KUKA KRL program: EPS_2_251825_SA26_A_20260116064103.src

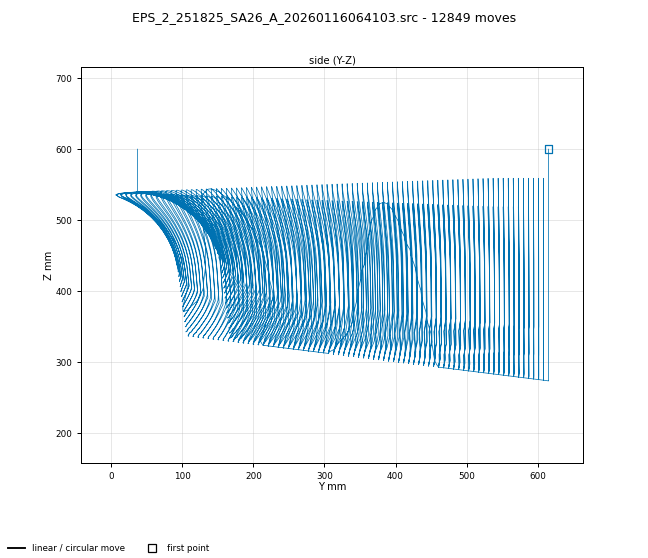
[picture p0: tool path of EPS_2_251825_SA26_A_20260116064103.src, 12849 of 12851 moves have a stored position in this frame; points joined in program order, loops and branches not executed]
&ACCESS RVP
&REL 4
&COMMENT QRS 19112012
&PARAM EDITMASK = *
DEF PART()
EXT BAS (BAS_COMMAND :IN,REAL :IN )
INT I
BAS (#INITMOV,0 )

;KUKA QRS Post kuka4.cps  Date:22-06-2017 !

File_ID=2985

QRS_PRE_INIT()

;Init var - Until changes are made in qrs_pre_init
Outlet_Square_prg=0
Inlet_1_Square_prg=0
Inlet_2_Square_prg=0
Inlet_3_Square_prg=0
Inlet_4_Square_prg=0
Inlet_5_Square_prg=0

Outlet_1={X 0.000, Y 535.490, Z 458.500, B 0.000, E1 0.000 }
Inlet_1={X 0.000, Y 538.340, Z 418.500, B 0.000, E1 190.000 }
Outlet_1_type=201
Inlet_1_type=201
;QRS#1=Sidecore dimensions
;QRS#2=200-8" PVC SDR 35
;QRS#3=200-8" PVC SDR 35
;QRS#4=
;QRS#5=
;QRS#6=
;QRS#7=
;QRS#8=
;QRS#9=12-08 PSX
;QRS#10=12-08 PSX
;QRS#11=
;QRS#12=
;QRS#13=
;QRS#14=
;QRS#15=
;QRS#16=1220x127x838 2,75'
;QRS#17=EPS Height
;QRS#18=559
;QRS#19=*
;QRS#20= UPDATED VERSION 22-06-2017
;QRS#21=*
Outlet_Square=0100
Inlet_1_Square=0100
Inlet_2_Square=0
Inlet_3_Square=0
Inlet_4_Square=0
Inlet_5_Square=0
Mill_Square=1
Outlet_Square_Prg=204
Inlet_1_Square_prg=204

QRS_INIT()

$ADVANCE=5

; T1
PTP {E1 173.626,E2 173.626}
PTP {X 0,Y 615.464,A -85,B 0,C 180,E1 173.626,E2 173.626,E3 0,E4 0,E5 0,E6 0}
QRS_SPEED_INIT()
LIN {X 0,Y 615.464,Z 600,A -85,B 0,C 180,E1 173.626,E2 173.626,E3 0,E4 0,E5 0,E6 0} C_VEL
LIN {X 0,Y 615.464,Z 283.872,A -85,B 0,C 180,E1 173.626,E2 173.626} C_VEL
LIN {X 0,Y 615.464,Z 275.69,A -85,B 0,C 180,E1 173.626,E2 173.626} C_VEL
LIN {X 0,Y 615.457,Z 273.69,A -85,B 0,C 180,E1 173.44,E2 173.44} C_VEL
LIN {X 0,Y 615.487,Z 273.682,A -85,B 0,C 180,E1 170.801,E2 170.801} C_VEL
LIN {X 0,Y 615.491,Z 273.695,A -85,B 0,C 180,E1 168.139,E2 168.139} C_VEL
LIN {X 0,Y 615.461,Z 273.694,A -85,B 0,C 180,E1 165.45,E2 165.45} C_VEL
LIN {X 0,Y 615.46,Z 273.695,A -85,B 0,C 180,E1 163.413,E2 163.413} C_VEL
LIN {X 0,Y 615.46,Z 273.694,A -85,B 0,C 180,E1 161.353,E2 161.353} C_VEL
LIN {X 0,Y 615.458,Z 273.694,A -85,B 0,C 180,E1 159.268,E2 159.268} C_VEL
LIN {X 0,Y 615.455,Z 273.694,A -85,B 0,C 180,E1 157.154,E2 157.154} C_VEL
LIN {X 0,Y 615.451,Z 273.693,A -85,B 0,C 180,E1 155.007,E2 155.007} C_VEL
LIN {X 0,Y 615.449,Z 273.691,A -85,B 0,C 180,E1 152.821,E2 152.821} C_VEL
LIN {X 0,Y 615.476,Z 273.685,A -85,B 0,C 180,E1 150.206,E2 150.206} C_VEL
LIN {X 0,Y 615.493,Z 273.695,A -85,B 0,C 180,E1 147.543,E2 147.543} C_VEL
LIN {X 0,Y 615.482,Z 273.698,A -85,B 0,C 180,E1 145.185,E2 145.185} C_VEL
LIN {X 0,Y 615.45,Z 273.695,A -85,B 0,C 180,E1 142.755,E2 142.755} C_VEL
LIN {X 0,Y 615.447,Z 273.69,A -85,B 0,C 180,E1 140.247,E2 140.247} C_VEL
LIN {X 0,Y 615.491,Z 273.685,A -85,B 0,C 180,E1 137.647,E2 137.647} C_VEL
LIN {X 0,Y 615.484,Z 273.699,A -85,B 0,C 180,E1 134.931,E2 134.931} C_VEL
LIN {X 0,Y 615.442,Z 273.694,A -85,B 0,C 180,E1 132.356,E2 132.356} C_VEL
LIN {X 0,Y 615.439,Z 273.692,A -85,B 0,C 180,E1 130.084,E2 130.084} C_VEL
LIN {X 0,Y 615.438,Z 273.692,A -85,B 0,C 180,E1 128.006,E2 128.006} C_VEL
LIN {X 0,Y 615.449,Z 273.69,A -85,B 0,C 180,E1 125.618,E2 125.618} C_VEL
LIN {X 0,Y 615.474,Z 273.689,A -85,B 0,C 180,E1 123.236,E2 123.236} C_VEL
LIN {X 0,Y 615.49,Z 273.692,A -85,B 0,C 180,E1 120.919,E2 120.919} C_VEL
LIN {X 0,Y 615.435,Z 273.695,A -85,B 0,C 180,E1 117.917,E2 117.917} C_VEL
LIN {X 0,Y 615.433,Z 273.693,A -85,B 0,C 180,E1 115.558,E2 115.558} C_VEL
LIN {X 0,Y 615.484,Z 273.689,A -85,B 0,C 180,E1 112.844,E2 112.844} C_VEL
LIN {X 0,Y 615.455,Z 273.698,A -85,B 0,C 180,E1 110.033,E2 110.033} C_VEL
LIN {X 0,Y 615.453,Z 273.698,A -85,B 0,C 180,E1 107.958,E2 107.958} C_VEL
LIN {X 0,Y 615.452,Z 273.698,A -85,B 0,C 180,E1 105.906,E2 105.906} C_VEL
LIN {X 0,Y 615.455,Z 273.698,A -85,B 0,C 180,E1 103.875,E2 103.875} C_VEL
LIN {X 0,Y 615.46,Z 273.699,A -85,B 0,C 180,E1 101.861,E2 101.861} C_VEL
LIN {X 0,Y 615.423,Z 273.696,A -85,B 0,C 180,E1 99.199,E2 99.199} C_VEL
LIN {X 0,Y 615.453,Z 273.715,A -85,B 0,C 180,E1 98.62,E2 98.62} C_VEL
LIN {X 0,Y 615.457,Z 289.755,A -85,B 0,C 180,E1 95.899,E2 95.899} C_VEL
LIN {X 0,Y 615.446,Z 303.472,A -85,B 0,C 180,E1 93.601,E2 93.601} C_VEL
LIN {X 0,Y 615.464,Z 308.129,A -85,B 0,C 180,E1 92.822,E2 92.822} C_VEL
LIN {X 0,Y 615.458,Z 415.467,A -85,B 0,C 180,E1 91.533,E2 91.533} C_VEL
LIN {X 0,Y 615.458,Z 429.062,A -85,B 0,C 180,E1 91.227,E2 91.227} C_VEL
LIN {X 0,Y 615.485,Z 441.275,A -85,B 0,C 180,E1 90.818,E2 90.818} C_VEL
LIN {X 0,Y 615.489,Z 452.256,A -85,B 0,C 180,E1 90.327,E2 90.327} C_VEL
LIN {X 0,Y 615.488,Z 463.666,A -85,B 0,C 180,E1 89.673,E2 89.673} C_VEL
LIN {X 0,Y 615.499,Z 473.94,A -85,B 0,C 180,E1 88.937,E2 88.937} C_VEL
LIN {X 0,Y 615.497,Z 482.288,A -85,B 0,C 180,E1 88.2,E2 88.2} C_VEL
LIN {X 0,Y 615.497,Z 490.195,A -85,B 0,C 180,E1 87.382,E2 87.382} C_VEL
LIN {X 0,Y 615.493,Z 497.851,A -85,B 0,C 180,E1 86.399,E2 86.399} C_VEL
LIN {X 0,Y 615.496,Z 504.004,A -85,B 0,C 180,E1 85.415,E2 85.415} C_VEL
LIN {X 0,Y 615.497,Z 508.911,A -85,B 0,C 180,E1 84.43,E2 84.43} C_VEL
LIN {X 0,Y 615.495,Z 512.797,A -85,B 0,C 180,E1 83.416,E2 83.416} C_VEL
LIN {X 0,Y 615.495,Z 516.218,A -85,B 0,C 180,E1 82.124,E2 82.124} C_VEL
LIN {X 0,Y 615.495,Z 517.345,A -85,B 0,C 180,E1 81.463,E2 81.463} C_VEL
LIN {X 0,Y 615.496,Z 518.351,A -85,B 0,C 180,E1 80.138,E2 80.138} C_VEL
LIN {X 0,Y 615.494,Z 518.038,A -85,B 0,C 180,E1 79.109,E2 79.109} C_VEL
LIN {X 0,Y 615.495,Z 516.853,A -85,B 0,C 180,E1 78.139,E2 78.139} C_VEL
LIN {X 0,Y 615.496,Z 515.533,A -85,B 0,C 180,E1 77.47,E2 77.47} C_VEL
LIN {X 0,Y 615.496,Z 512.696,A -85,B 0,C 180,E1 76.463,E2 76.463} C_VEL
LIN {X 0,Y 615.497,Z 508.787,A -85,B 0,C 180,E1 75.451,E2 75.451} C_VEL
LIN {X 0,Y 615.496,Z 503.676,A -85,B 0,C 180,E1 74.435,E2 74.435} C_VEL
LIN {X 0,Y 615.495,Z 497.179,A -85,B 0,C 180,E1 73.414,E2 73.414} C_VEL
LIN {X 0,Y 615.498,Z 488.929,A -85,B 0,C 180,E1 72.387,E2 72.387} C_VEL
LIN {X 0,Y 615.497,Z 478.509,A -85,B 0,C 180,E1 71.354,E2 71.354} C_VEL
LIN {X 0,Y 615.494,Z 467.446,A -85,B 0,C 180,E1 70.489,E2 70.489} C_VEL
LIN {X 0,Y 615.465,Z 457.023,A -85,B 0,C 180,E1 69.836,E2 69.836} C_VEL
LIN {X 0,Y 615.492,Z 445.516,A -85,B 0,C 180,E1 69.269,E2 69.269} C_VEL
LIN {X 0,Y 615.443,Z 432.543,A -85,B 0,C 180,E1 68.786,E2 68.786} C_VEL
LIN {X 0,Y 615.424,Z 419.82,A -85,B 0,C 180,E1 68.456,E2 68.456} C_VEL
LIN {X 0,Y 615.422,Z 405.107,A -85,B 0,C 180,E1 68.236,E2 68.236} C_VEL
LIN {X 0,Y 615.476,Z 308.131,A -85,B 0,C 180,E1 67.088,E2 67.088} C_VEL
LIN {X 0,Y 615.45,Z 292.299,A -85,B 0,C 180,E1 64.438,E2 64.438} C_VEL
LIN {X 0,Y 615.494,Z 276.796,A -85,B 0,C 180,E1 61.818,E2 61.818} C_VEL
LIN {X 0,Y 615.488,Z 273.684,A -85,B 0,C 180,E1 61.249,E2 61.249} C_VEL
LIN {X 0,Y 615.483,Z 273.682,A -85,B 0,C 180,E1 58.915,E2 58.915} C_VEL
LIN {X 0,Y 615.469,Z 273.686,A -85,B 0,C 180,E1 56.468,E2 56.468} C_VEL
LIN {X 0,Y 615.466,Z 273.69,A -85,B 0,C 180,E1 54.169,E2 54.169} C_VEL
LIN {X 0,Y 615.471,Z 273.693,A -85,B 0,C 180,E1 51.93,E2 51.93} C_VEL
LIN {X 0,Y 615.493,Z 273.698,A -85,B 0,C 180,E1 49.394,E2 49.394} C_VEL
LIN {X 0,Y 615.487,Z 273.683,A -85,B 0,C 180,E1 46.755,E2 46.755} C_VEL
LIN {X 0,Y 615.469,Z 273.687,A -85,B 0,C 180,E1 43.996,E2 43.996} C_VEL
LIN {X 0,Y 615.479,Z 273.696,A -85,B 0,C 180,E1 41.474,E2 41.474} C_VEL
LIN {X 0,Y 615.484,Z 273.694,A -85,B 0,C 180,E1 38.904,E2 38.904} C_VEL
LIN {X 0,Y 615.486,Z 273.683,A -85,B 0,C 180,E1 36.425,E2 36.425} C_VEL
LIN {X 0,Y 615.489,Z 273.68,A -85,B 0,C 180,E1 34.022,E2 34.022} C_VEL
LIN {X 0,Y 615.48,Z 273.698,A -85,B 0,C 180,E1 31.085,E2 31.085} C_VEL
LIN {X 0,Y 615.48,Z 273.69,A -85,B 0,C 180,E1 28.449,E2 28.449} C_VEL
LIN {X 0,Y 615.477,Z 273.684,A -85,B 0,C 180,E1 25.567,E2 25.567} C_VEL
LIN {X 0,Y 615.484,Z 273.697,A -85,B 0,C 180,E1 22.845,E2 22.845} C_VEL
LIN {X 0,Y 615.48,Z 273.687,A -85,B 0,C 180,E1 20.033,E2 20.033} C_VEL
LIN {X 0,Y 615.474,Z 273.685,A -85,B 0,C 180,E1 17.271,E2 17.271} C_VEL
LIN {X 0,Y 615.488,Z 273.697,A -85,B 0,C 180,E1 14.549,E2 14.549} C_VEL
LIN {X 0,Y 615.478,Z 273.689,A -85,B 0,C 180,E1 11.861,E2 11.861} C_VEL
LIN {X 0,Y 615.49,Z 273.68,A -85,B 0,C 180,E1 9.199,E2 9.199} C_VEL
LIN {X 0,Y 615.474,Z 273.692,A -85,B 0,C 180,E1 6.557,E2 6.557} C_VEL
LIN {X 0,Y 615.488,Z 273.696,A -85,B 0,C 180,E1 3.928,E2 3.928} C_VEL
LIN {X 0,Y 615.482,Z 273.684,A -85,B 0,C 180,E1 1.308,E2 1.308} C_VEL
LIN {X 0,Y 615.48,Z 273.683,A -85,B 0,C 180,E1 -1.309,E2 -1.309} C_VEL
LIN {X 0,Y 615.482,Z 273.695,A -85,B 0,C 180,E1 -3.929,E2 -3.929} C_VEL
LIN {X 0,Y 615.475,Z 273.693,A -85,B 0,C 180,E1 -6.57,E2 -6.57} C_VEL
LIN {X 0,Y 615.491,Z 273.68,A -85,B 0,C 180,E1 -9.199,E2 -9.199} C_VEL
LIN {X 0,Y 615.475,Z 273.688,A -85,B 0,C 180,E1 -11.861,E2 -11.861} C_VEL
LIN {X 0,Y 615.492,Z 273.699,A -85,B 0,C 180,E1 -14.549,E2 -14.549} C_VEL
LIN {X 0,Y 615.476,Z 273.685,A -85,B 0,C 180,E1 -17.271,E2 -17.271} C_VEL
LIN {X 0,Y 615.478,Z 273.686,A -85,B 0,C 180,E1 -20.033,E2 -20.033} C_VEL
LIN {X 0,Y 615.49,Z 273.698,A -85,B 0,C 180,E1 -22.845,E2 -22.845} C_VEL
LIN {X 0,Y 615.488,Z 273.681,A -85,B 0,C 180,E1 -25.716,E2 -25.716} C_VEL
LIN {X 0,Y 615.477,Z 273.689,A -85,B 0,C 180,E1 -28.449,E2 -28.449} C_VEL
LIN {X 0,Y 615.482,Z 273.7,A -85,B 0,C 180,E1 -31.086,E2 -31.086} C_VEL
LIN {X 0,Y 615.49,Z 273.68,A -85,B 0,C 180,E1 -34.022,E2 -34.022} C_VEL
LIN {X 0,Y 615.484,Z 273.695,A -85,B 0,C 180,E1 -36.936,E2 -36.936} C_VEL
LIN {X 0,Y 615.472,Z 273.69,A -85,B 0,C 180,E1 -39.752,E2 -39.752} C_VEL
LIN {X 0,Y 615.493,Z 273.679,A -85,B 0,C 180,E1 -42.353,E2 -42.353} C_VEL
LIN {X 0,Y 615.477,Z 273.692,A -85,B 0,C 180,E1 -45.07,E2 -45.07} C_VEL
LIN {X 0,Y 615.469,Z 273.692,A -85,B 0,C 180,E1 -47.922,E2 -47.922} C_VEL
LIN {X 0,Y 615.472,Z 273.686,A -85,B 0,C 180,E1 -50.249,E2 -50.249} C_VEL
LIN {X 0,Y 615.481,Z 273.685,A -85,B 0,C 180,E1 -53.065,E2 -53.065} C_VEL
LIN {X 0,Y 615.481,Z 273.696,A -85,B 0,C 180,E1 -55.978,E2 -55.978} C_VEL
LIN {X 0,Y 615.47,Z 273.69,A -85,B 0,C 180,E1 -58.314,E2 -58.314} C_VEL
LIN {X 0,Y 615.471,Z 273.686,A -85,B 0,C 180,E1 -60.593,E2 -60.593} C_VEL
LIN {X 0,Y 615.486,Z 273.681,A -85,B 0,C 180,E1 -62.956,E2 -62.956} C_VEL
LIN {X 0,Y 615.481,Z 273.692,A -85,B 0,C 180,E1 -65.728,E2 -65.728} C_VEL
LIN {X 0,Y 615.487,Z 273.754,A -85,B 0,C 180,E1 -67.437,E2 -67.437} C_VEL
LIN {X 0,Y 615.455,Z 293.691,A -85,B 0,C 180,E1 -70.14,E2 -70.14} C_VEL
LIN {X 0,Y 615.472,Z 313.076,A -85,B 0,C 180,E1 -72.729,E2 -72.729} C_VEL
LIN {X 0,Y 615.493,Z 334.916,A -85,B 0,C 180,E1 -75.606,E2 -75.606} C_VEL
LIN {X 0,Y 615.471,Z 346.467,A -85,B 0,C 180,E1 -77.113,E2 -77.113} C_VEL
LIN {X 0,Y 615.457,Z 454.829,A -85,B 0,C 180,E1 -78.41,E2 -78.41} C_VEL
LIN {X 0,Y 615.456,Z 467.345,A -85,B 0,C 180,E1 -78.681,E2 -78.681} C_VEL
LIN {X 0,Y 615.483,Z 480.688,A -85,B 0,C 180,E1 -79.116,E2 -79.116} C_VEL
LIN {X 0,Y 615.492,Z 492.473,A -85,B 0,C 180,E1 -79.639,E2 -79.639} C_VEL
LIN {X 0,Y 615.483,Z 503.994,A -85,B 0,C 180,E1 -80.304,E2 -80.304} C_VEL
LIN {X 0,Y 615.499,Z 514.339,A -85,B 0,C 180,E1 -81.05,E2 -81.05} C_VEL
LIN {X 0,Y 615.497,Z 522.69,A -85,B 0,C 180,E1 -81.794,E2 -81.794} C_VEL
LIN {X 0,Y 615.498,Z 530.605,A -85,B 0,C 180,E1 -82.619,E2 -82.619} C_VEL
LIN {X 0,Y 615.491,Z 538.203,A -85,B 0,C 180,E1 -83.608,E2 -83.608} C_VEL
LIN {X 0,Y 615.498,Z 545.203,A -85,B 0,C 180,E1 -84.759,E2 -84.759} C_VEL
LIN {X 0,Y 615.493,Z 549.851,A -85,B 0,C 180,E1 -85.743,E2 -85.743} C_VEL
LIN {X 0,Y 615.494,Z 553.398,A -85,B 0,C 180,E1 -86.727,E2 -86.727} C_VEL
LIN {X 0,Y 615.497,Z 555.232,A -85,B 0,C 180,E1 -87.382,E2 -87.382} C_VEL
LIN {X 0,Y 615.497,Z 556.608,A -85,B 0,C 180,E1 -88.037,E2 -88.037} C_VEL
LIN {X 0,Y 615.496,Z 558.173,A -85,B 0,C 180,E1 -89.346,E2 -89.346} C_VEL
LIN {X 0,Y 615.494,Z 558.389,A -85,B 0,C 180,E1 -90,E2 -90} C_VEL
LIN {X 0,Y 615.495,Z 557.58,A -85,B 0,C 180,E1 -91.308,E2 -91.308} C_VEL
LIN {X 0,Y 615.497,Z 556.609,A -85,B 0,C 180,E1 -91.963,E2 -91.963} C_VEL
LIN {X 0,Y 615.497,Z 555.234,A -85,B 0,C 180,E1 -92.618,E2 -92.618} C_VEL
LIN {X 0,Y 615.496,Z 552.35,A -85,B 0,C 180,E1 -93.6,E2 -93.6} C_VEL
LIN {X 0,Y 615.498,Z 548.443,A -85,B 0,C 180,E1 -94.584,E2 -94.584} C_VEL
LIN {X 0,Y 615.499,Z 543.406,A -85,B 0,C 180,E1 -95.569,E2 -95.569} C_VEL
LIN {X 0,Y 615.49,Z 536.913,A -85,B 0,C 180,E1 -96.578,E2 -96.578} C_VEL
LIN {X 0,Y 615.497,Z 529.136,A -85,B 0,C 180,E1 -97.545,E2 -97.545} C_VEL
LIN {X 0,Y 615.498,Z 519.261,A -85,B 0,C 180,E1 -98.536,E2 -98.536} C_VEL
LIN {X 0,Y 615.495,Z 508.87,A -85,B 0,C 180,E1 -99.364,E2 -99.364} C_VEL
LIN {X 0,Y 615.482,Z 498.581,A -85,B 0,C 180,E1 -100.028,E2 -100.028} C_VEL
LIN {X 0,Y 615.495,Z 487.142,A -85,B 0,C 180,E1 -100.616,E2 -100.616} C_VEL
LIN {X 0,Y 615.467,Z 475.364,A -85,B 0,C 180,E1 -101.077,E2 -101.077} C_VEL
LIN {X 0,Y 615.455,Z 462.262,A -85,B 0,C 180,E1 -101.444,E2 -101.444} C_VEL
LIN {X 0,Y 615.461,Z 448.976,A -85,B 0,C 180,E1 -101.673,E2 -101.673} C_VEL
LIN {X 0,Y 615.471,Z 346.471,A -85,B 0,C 180,E1 -102.886,E2 -102.886} C_VEL
LIN {X 0,Y 615.455,Z 325.993,A -85,B 0,C 180,E1 -105.566,E2 -105.566} C_VEL
LIN {X 0,Y 615.481,Z 305.476,A -85,B 0,C 180,E1 -108.281,E2 -108.281} C_VEL
LIN {X 0,Y 615.468,Z 283.347,A -85,B 0,C 180,E1 -111.257,E2 -111.257} C_VEL
LIN {X 0,Y 615.489,Z 273.682,A -85,B 0,C 180,E1 -112.594,E2 -112.594} C_VEL
LIN {X 0,Y 615.485,Z 273.681,A -85,B 0,C 180,E1 -114.991,E2 -114.991} C_VEL
LIN {X 0,Y 615.482,Z 273.699,A -85,B 0,C 180,E1 -117.915,E2 -117.915} C_VEL
LIN {X 0,Y 615.485,Z 273.682,A -85,B 0,C 180,E1 -120.919,E2 -120.919} C_VEL
LIN {X 0,Y 615.473,Z 273.686,A -85,B 0,C 180,E1 -123.532,E2 -123.532} C_VEL
LIN {X 0,Y 615.488,Z 273.696,A -85,B 0,C 180,E1 -126.424,E2 -126.424} C_VEL
LIN {X 0,Y 615.48,Z 273.684,A -85,B 0,C 180,E1 -129.061,E2 -129.061} C_VEL
LIN {X 0,Y 615.492,Z 273.68,A -85,B 0,C 180,E1 -131.473,E2 -131.473} C_VEL
LIN {X 0,Y 615.477,Z 273.693,A -85,B 0,C 180,E1 -134.15,E2 -134.15} C_VEL
LIN {X 0,Y 615.476,Z 273.691,A -85,B 0,C 180,E1 -136.953,E2 -136.953} C_VEL
LIN {X 0,Y 615.481,Z 273.683,A -85,B 0,C 180,E1 -139.393,E2 -139.393} C_VEL
LIN {X 0,Y 615.482,Z 273.684,A -85,B 0,C 180,E1 -141.988,E2 -141.988} C_VEL
LIN {X 0,Y 615.479,Z 273.691,A -85,B 0,C 180,E1 -144.383,E2 -144.383} C_VEL
LIN {X 0,Y 615.484,Z 273.701,A -85,B 0,C 180,E1 -146.763,E2 -146.763} C_VEL
LIN {X 0,Y 615.48,Z 273.697,A -85,B 0,C 180,E1 -149.08,E2 -149.08} C_VEL
LIN {X 0,Y 615.47,Z 273.688,A -85,B 0,C 180,E1 -151.551,E2 -151.551} C_VEL
LIN {X 0,Y 615.49,Z 273.682,A -85,B 0,C 180,E1 -154.284,E2 -154.284} C_VEL
LIN {X 0,Y 615.484,Z 273.701,A -85,B 0,C 180,E1 -157.155,E2 -157.155} C_VEL
LIN {X 0,Y 615.472,Z 273.685,A -85,B 0,C 180,E1 -159.967,E2 -159.967} C_VEL
LIN {X 0,Y 615.482,Z 273.687,A -85,B 0,C 180,E1 -162.729,E2 -162.729} C_VEL
LIN {X 0,Y 615.482,Z 273.699,A -85,B 0,C 180,E1 -165.451,E2 -165.451} C_VEL
LIN {X 0,Y 615.464,Z 273.687,A -85,B 0,C 180,E1 -168.139,E2 -168.139} C_VEL
LIN {X 0,Y 615.493,Z 273.682,A -85,B 0,C 180,E1 -170.801,E2 -170.801} C_VEL
LIN {X 0,Y 615.493,Z 273.697,A -85,B 0,C 180,E1 -173.443,E2 -173.443} C_VEL
LIN {X 0,Y 615.464,Z 273.693,A -85,B 0,C 180,E1 -176.071,E2 -176.071} C_VEL
LIN {X 0,Y 615.474,Z 273.684,A -85,B 0,C 180,E1 -178.691,E2 -178.691} C_VEL
LIN {X 0,Y 615.488,Z 273.687,A -85,B 0,C 180,E1 -181.308,E2 -181.308} C_VEL
LIN {X 0,Y 615.483,Z 273.7,A -85,B 0,C 180,E1 -183.928,E2 -183.928} C_VEL
LIN {X 0,Y 615.457,Z 273.69,A -85,B 0,C 180,E1 -186.56,E2 -186.56} C_VEL
LIN {X 0,Y 614.8,Z 273.833,A -85,B 0,C 180,E1 -187.106,E2 -187.106} C_VEL
LIN {X 0,Y 611.98,Z 274.258,A -85,B 0,C 180,E1 -187.992,E2 -187.992} C_VEL
LIN {X 0,Y 609.59,Z 274.561,A -85,B 0,C 180,E1 -188.705,E2 -188.705} C_VEL
LIN {X 0,Y 608.552,Z 274.677,A -85,B 0,C 180,E1 -189.255,E2 -189.255} C_VEL
LIN {X 0,Y 608.461,Z 274.688,A -85,B 0,C 180,E1 -189.441,E2 -189.441} C_VEL
LIN {X 0,Y 608.459,Z 274.696,A -85,B 0,C 180,E1 -192,E2 -192} C_VEL
LIN {X 0,Y 608.426,Z 274.692,A -85,B 0,C 180,E1 -194.722,E2 -194.722} C_VEL
LIN {X 0,Y 608.426,Z 274.692,A -85,B 0,C 180,E1 -196.785,E2 -196.785} C_VEL
LIN {X 0,Y 608.442,Z 274.689,A -85,B 0,C 180,E1 -199.571,E2 -199.571} C_VEL
LIN {X 0,Y 608.452,Z 274.695,A -85,B 0,C 180,E1 -202.477,E2 -202.477} C_VEL
LIN {X 0,Y 608.444,Z 274.696,A -85,B 0,C 180,E1 -204.571,E2 -204.571} C_VEL
LIN {X 0,Y 608.427,Z 274.69,A -85,B 0,C 180,E1 -207.199,E2 -207.199} C_VEL
LIN {X 0,Y 608.46,Z 274.686,A -85,B 0,C 180,E1 -209.78,E2 -209.78} C_VEL
LIN {X 0,Y 608.465,Z 274.695,A -85,B 0,C 180,E1 -212.524,E2 -212.524} C_VEL
LIN {X 0,Y 608.421,Z 274.692,A -85,B 0,C 180,E1 -215.279,E2 -215.279} C_VEL
LIN {X 0,Y 608.448,Z 274.687,A -85,B 0,C 180,E1 -217.748,E2 -217.748} C_VEL
LIN {X 0,Y 608.444,Z 274.69,A -85,B 0,C 180,E1 -220.329,E2 -220.329} C_VEL
LIN {X 0,Y 608.45,Z 274.691,A -85,B 0,C 180,E1 -223.308,E2 -223.308} C_VEL
LIN {X 0,Y 608.44,Z 274.688,A -85,B 0,C 180,E1 -226.129,E2 -226.129} C_VEL
LIN {X 0,Y 608.462,Z 274.692,A -85,B 0,C 180,E1 -228.825,E2 -228.825} C_VEL
LIN {X 0,Y 608.433,Z 274.69,A -85,B 0,C 180,E1 -231.764,E2 -231.764} C_VEL
LIN {X 0,Y 608.427,Z 274.69,A -85,B 0,C 180,E1 -233.957,E2 -233.957} C_VEL
LIN {X 0,Y 608.439,Z 274.688,A -85,B 0,C 180,E1 -236.328,E2 -236.328} C_VEL
LIN {X 0,Y 608.439,Z 274.69,A -85,B 0,C 180,E1 -238.734,E2 -238.734} C_VEL
LIN {X 0,Y 608.428,Z 274.695,A -85,B 0,C 180,E1 -241.733,E2 -241.733} C_VEL
LIN {X 0,Y 608.428,Z 274.69,A -85,B 0,C 180,E1 -244.288,E2 -244.288} C_VEL
LIN {X 0,Y 608.429,Z 274.691,A -85,B 0,C 180,E1 -246.876,E2 -246.876} C_VEL
LIN {X 0,Y 608.45,Z 274.697,A -85,B 0,C 180,E1 -249.726,E2 -249.726} C_VEL
LIN {X 0,Y 608.429,Z 274.698,A -85,B 0,C 180,E1 -251.828,E2 -251.828} C_VEL
LIN {X 0,Y 608.442,Z 274.696,A -85,B 0,C 180,E1 -253.906,E2 -253.906} C_VEL
LIN {X 0,Y 608.431,Z 274.697,A -85,B 0,C 180,E1 -255.997,E2 -255.997} C_VEL
LIN {X 0,Y 608.442,Z 274.697,A -85,B 0,C 180,E1 -258,E2 -258} C_VEL
LIN {X 0,Y 608.419,Z 274.692,A -85,B 0,C 180,E1 -260.694,E2 -260.694} C_VEL
LIN {X 0,Y 608.425,Z 274.736,A -85,B 0,C 180,E1 -261.322,E2 -261.322} C_VEL
LIN {X 0,Y 608.465,Z 290.578,A -85,B 0,C 180,E1 -264.033,E2 -264.033} C_VEL
LIN {X 0,Y 608.407,Z 306.319,A -85,B 0,C 180,E1 -266.689,E2 -266.689} C_VEL
LIN {X 0,Y 608.422,Z 308.417,A -85,B 0,C 180,E1 -267.041,E2 -267.041} C_VEL
LIN {X 0,Y 608.532,Z 415.148,A -85,B 0,C 180,E1 -268.325,E2 -268.325} C_VEL
LIN {X 0,Y 608.516,Z 428.146,A -85,B 0,C 180,E1 -268.615,E2 -268.615} C_VEL
LIN {X 0,Y 608.52,Z 441.205,A -85,B 0,C 180,E1 -269.049,E2 -269.049} C_VEL
LIN {X 0,Y 608.503,Z 453.059,A -85,B 0,C 180,E1 -269.587,E2 -269.587} C_VEL
LIN {X 0,Y 608.475,Z 464.387,A -85,B 0,C 180,E1 -270.248,E2 -270.248} C_VEL
LIN {X 0,Y 608.478,Z 475.661,A -85,B 0,C 180,E1 -271.076,E2 -271.076} C_VEL
LIN {X 0,Y 608.467,Z 483.782,A -85,B 0,C 180,E1 -271.82,E2 -271.82} C_VEL
LIN {X 0,Y 608.464,Z 491.538,A -85,B 0,C 180,E1 -272.648,E2 -272.648} C_VEL
LIN {X 0,Y 608.448,Z 499.048,A -85,B 0,C 180,E1 -273.643,E2 -273.643} C_VEL
LIN {X 0,Y 608.445,Z 505.107,A -85,B 0,C 180,E1 -274.638,E2 -274.638} C_VEL
LIN {X 0,Y 608.43,Z 509.924,A -85,B 0,C 180,E1 -275.635,E2 -275.635} C_VEL
LIN {X 0,Y 608.444,Z 513.633,A -85,B 0,C 180,E1 -276.633,E2 -276.633} C_VEL
LIN {X 0,Y 608.423,Z 515.553,A -85,B 0,C 180,E1 -277.3,E2 -277.3} C_VEL
LIN {X 0,Y 608.422,Z 517.047,A -85,B 0,C 180,E1 -277.968,E2 -277.968} C_VEL
LIN {X 0,Y 608.421,Z 518.73,A -85,B 0,C 180,E1 -279.307,E2 -279.307} C_VEL
LIN {X 0,Y 608.432,Z 518.99,A -85,B 0,C 180,E1 -279.978,E2 -279.978} C_VEL
LIN {X 0,Y 608.421,Z 518.625,A -85,B 0,C 180,E1 -280.932,E2 -280.932} C_VEL
LIN {X 0,Y 608.44,Z 517.252,A -85,B 0,C 180,E1 -282,E2 -282} C_VEL
LIN {X 0,Y 608.423,Z 515.847,A -85,B 0,C 180,E1 -282.678,E2 -282.678} C_VEL
LIN {X 0,Y 608.429,Z 512.915,A -85,B 0,C 180,E1 -283.682,E2 -283.682} C_VEL
LIN {X 0,Y 608.432,Z 508.779,A -85,B 0,C 180,E1 -284.722,E2 -284.722} C_VEL
LIN {X 0,Y 608.461,Z 502.414,A -85,B 0,C 180,E1 -285.922,E2 -285.922} C_VEL
LIN {X 0,Y 608.461,Z 495.4,A -85,B 0,C 180,E1 -286.957,E2 -286.957} C_VEL
LIN {X 0,Y 608.457,Z 488.18,A -85,B 0,C 180,E1 -287.824,E2 -287.824} C_VEL
LIN {X 0,Y 608.47,Z 477.355,A -85,B 0,C 180,E1 -288.869,E2 -288.869} C_VEL
LIN {X 0,Y 608.472,Z 467.158,A -85,B 0,C 180,E1 -289.658,E2 -289.658} C_VEL
LIN {X 0,Y 608.467,Z 456.11,A -85,B 0,C 180,E1 -290.34,E2 -290.34} C_VEL
LIN {X 0,Y 608.522,Z 443.999,A -85,B 0,C 180,E1 -290.925,E2 -290.925} C_VEL
LIN {X 0,Y 608.479,Z 431.532,A -85,B 0,C 180,E1 -291.38,E2 -291.38} C_VEL
LIN {X 0,Y 608.481,Z 419.192,A -85,B 0,C 180,E1 -291.691,E2 -291.691} C_VEL
LIN {X 0,Y 608.497,Z 404.07,A -85,B 0,C 180,E1 -291.913,E2 -291.913} C_VEL
LIN {X 0,Y 608.476,Z 308.697,A -85,B 0,C 180,E1 -293.043,E2 -293.043} C_VEL
LIN {X 0,Y 608.429,Z 306.888,A -85,B 0,C 180,E1 -293.305,E2 -293.305} C_VEL
LIN {X 0,Y 608.444,Z 292.59,A -85,B 0,C 180,E1 -295.716,E2 -295.716} C_VEL
LIN {X 0,Y 608.497,Z 276.602,A -85,B 0,C 180,E1 -298.444,E2 -298.444} C_VEL
LIN {X 0,Y 608.483,Z 274.685,A -85,B 0,C 180,E1 -298.784,E2 -298.784} C_VEL
LIN {X 0,Y 608.442,Z 274.688,A -85,B 0,C 180,E1 -301.318,E2 -301.318} C_VEL
LIN {X 0,Y 608.445,Z 274.69,A -85,B 0,C 180,E1 -303.731,E2 -303.731} C_VEL
LIN {X 0,Y 608.442,Z 274.694,A -85,B 0,C 180,E1 -306.092,E2 -306.092} C_VEL
LIN {X 0,Y 608.462,Z 274.694,A -85,B 0,C 180,E1 -308.588,E2 -308.588} C_VEL
LIN {X 0,Y 608.464,Z 274.685,A -85,B 0,C 180,E1 -311.343,E2 -311.343} C_VEL
LIN {X 0,Y 608.441,Z 274.693,A -85,B 0,C 180,E1 -314.262,E2 -314.262} C_VEL
LIN {X 0,Y 608.453,Z 274.692,A -85,B 0,C 180,E1 -317.04,E2 -317.04} C_VEL
LIN {X 0,Y 608.451,Z 274.687,A -85,B 0,C 180,E1 -319.697,E2 -319.697} C_VEL
LIN {X 0,Y 608.465,Z 274.686,A -85,B 0,C 180,E1 -322.254,E2 -322.254} C_VEL
LIN {X 0,Y 608.449,Z 274.696,A -85,B 0,C 180,E1 -325.094,E2 -325.094} C_VEL
LIN {X 0,Y 608.462,Z 274.685,A -85,B 0,C 180,E1 -327.905,E2 -327.905} C_VEL
LIN {X 0,Y 608.467,Z 274.684,A -85,B 0,C 180,E1 -330.221,E2 -330.221} C_VEL
LIN {X 0,Y 608.47,Z 274.688,A -85,B 0,C 180,E1 -332.794,E2 -332.794} C_VEL
LIN {X 0,Y 608.447,Z 274.696,A -85,B 0,C 180,E1 -335.429,E2 -335.429} C_VEL
LIN {X 0,Y 608.462,Z 274.685,A -85,B 0,C 180,E1 -338.308,E2 -338.308} C_VEL
LIN {X 0,Y 608.474,Z 274.692,A -85,B 0,C 180,E1 -341.283,E2 -341.283} C_VEL
LIN {X 0,Y 608.457,Z 274.69,A -85,B 0,C 180,E1 -343.906,E2 -343.906} C_VEL
LIN {X 0,Y 608.458,Z 274.686,A -85,B 0,C 180,E1 -346.644,E2 -346.644} C_VEL
LIN {X 0,Y 608.457,Z 274.691,A -85,B 0,C 180,E1 -349.35,E2 -349.35} C_VEL
LIN {X 0,Y 608.472,Z 274.691,A -85,B 0,C 180,E1 -352.033,E2 -352.033} C_VEL
LIN {X 0,Y 608.467,Z 274.685,A -85,B 0,C 180,E1 -354.698,E2 -354.698} C_VEL
LIN {X 0,Y 608.466,Z 274.686,A -85,B 0,C 180,E1 -357.352,E2 -357.352} C_VEL
LIN {X 0,Y 608.476,Z 274.695,A -85,B 0,C 180,E1 -360,E2 -360} C_VEL
LIN {X 0,Y 608.469,Z 274.687,A -85,B 0,C 180,E1 -362.648,E2 -362.648} C_VEL
LIN {X 0,Y 608.467,Z 274.685,A -85,B 0,C 180,E1 -365.302,E2 -365.302} C_VEL
LIN {X 0,Y 608.468,Z 274.69,A -85,B 0,C 180,E1 -367.967,E2 -367.967} C_VEL
LIN {X 0,Y 608.461,Z 274.691,A -85,B 0,C 180,E1 -370.65,E2 -370.65} C_VEL
LIN {X 0,Y 608.459,Z 274.686,A -85,B 0,C 180,E1 -373.357,E2 -373.357} C_VEL
LIN {X 0,Y 608.455,Z 274.69,A -85,B 0,C 180,E1 -376.094,E2 -376.094} C_VEL
LIN {X 0,Y 608.456,Z 274.693,A -85,B 0,C 180,E1 -378.87,E2 -378.87} C_VEL
LIN {X 0,Y 608.459,Z 274.685,A -85,B 0,C 180,E1 -381.692,E2 -381.692} C_VEL
LIN {X 0,Y 608.448,Z 274.694,A -85,B 0,C 180,E1 -384.571,E2 -384.571} C_VEL
LIN {X 0,Y 608.474,Z 274.689,A -85,B 0,C 180,E1 -387.207,E2 -387.207} C_VEL
LIN {X 0,Y 608.466,Z 274.685,A -85,B 0,C 180,E1 -389.972,E2 -389.972} C_VEL
LIN {X 0,Y 608.452,Z 274.695,A -85,B 0,C 180,E1 -392.88,E2 -392.88} C_VEL
LIN {X 0,Y 608.434,Z 274.697,A -85,B 0,C 180,E1 -395.278,E2 -395.278} C_VEL
LIN {X 0,Y 608.467,Z 274.687,A -85,B 0,C 180,E1 -397.747,E2 -397.747} C_VEL
LIN {X 0,Y 608.446,Z 274.687,A -85,B 0,C 180,E1 -400.329,E2 -400.329} C_VEL
LIN {X 0,Y 608.477,Z 274.694,A -85,B 0,C 180,E1 -403.31,E2 -403.31} C_VEL
LIN {X 0,Y 608.459,Z 274.687,A -85,B 0,C 180,E1 -406.13,E2 -406.13} C_VEL
LIN {X 0,Y 608.454,Z 274.687,A -85,B 0,C 180,E1 -408.823,E2 -408.823} C_VEL
LIN {X 0,Y 608.46,Z 274.695,A -85,B 0,C 180,E1 -411.761,E2 -411.761} C_VEL
LIN {X 0,Y 608.444,Z 274.694,A -85,B 0,C 180,E1 -413.955,E2 -413.955} C_VEL
LIN {X 0,Y 608.444,Z 274.69,A -85,B 0,C 180,E1 -416.328,E2 -416.328} C_VEL
LIN {X 0,Y 608.446,Z 274.687,A -85,B 0,C 180,E1 -418.733,E2 -418.733} C_VEL
LIN {X 0,Y 608.47,Z 274.687,A -85,B 0,C 180,E1 -421.381,E2 -421.381} C_VEL
LIN {X 0,Y 608.438,Z 274.699,A -85,B 0,C 180,E1 -423.964,E2 -423.964} C_VEL
LIN {X 0,Y 608.464,Z 274.696,A -85,B 0,C 180,E1 -426.155,E2 -426.155} C_VEL
LIN {X 0,Y 608.507,Z 274.82,A -85,B 0,C 180,E1 -427.312,E2 -427.312} C_VEL
LIN {X 0,Y 608.524,Z 292.406,A -85,B 0,C 180,E1 -429.728,E2 -429.728} C_VEL
LIN {X 0,Y 608.51,Z 311.823,A -85,B 0,C 180,E1 -432.352,E2 -432.352} C_VEL
LIN {X 0,Y 608.496,Z 332.535,A -85,B 0,C 180,E1 -435.109,E2 -435.109} C_VEL
LIN {X 0,Y 608.454,Z 346.612,A -85,B 0,C 180,E1 -436.962,E2 -436.962} C_VEL
LIN {X 0,Y 608.575,Z 391.849,A -85,B 0,C 180,E1 -437.516,E2 -437.516} C_VEL
LIN {X 0,Y 608.522,Z 454.939,A -85,B 0,C 180,E1 -438.276,E2 -438.276} C_VEL
LIN {X 0,Y 608.491,Z 468.211,A -85,B 0,C 180,E1 -438.571,E2 -438.571} C_VEL
LIN {X 0,Y 608.511,Z 480.652,A -85,B 0,C 180,E1 -438.983,E2 -438.983} C_VEL
LIN {X 0,Y 608.514,Z 492.632,A -85,B 0,C 180,E1 -439.519,E2 -439.519} C_VEL
LIN {X 0,Y 608.471,Z 504.195,A -85,B 0,C 180,E1 -440.191,E2 -440.191} C_VEL
LIN {X 0,Y 608.485,Z 514.592,A -85,B 0,C 180,E1 -440.946,E2 -440.946} C_VEL
LIN {X 0,Y 608.459,Z 523,A -85,B 0,C 180,E1 -441.698,E2 -441.698} C_VEL
LIN {X 0,Y 608.471,Z 530.959,A -85,B 0,C 180,E1 -442.534,E2 -442.534} C_VEL
LIN {X 0,Y 608.436,Z 538.298,A -85,B 0,C 180,E1 -443.486,E2 -443.486} C_VEL
LIN {X 0,Y 608.45,Z 543.865,A -85,B 0,C 180,E1 -444.365,E2 -444.365} C_VEL
LIN {X 0,Y 608.432,Z 548.949,A -85,B 0,C 180,E1 -445.362,E2 -445.362} C_VEL
LIN {X 0,Y 608.449,Z 552.895,A -85,B 0,C 180,E1 -446.357,E2 -446.357} C_VEL
LIN {X 0,Y 608.425,Z 555.808,A -85,B 0,C 180,E1 -447.352,E2 -447.352} C_VEL
LIN {X 0,Y 608.442,Z 557.201,A -85,B 0,C 180,E1 -448.014,E2 -448.014} C_VEL
LIN {X 0,Y 608.439,Z 558.783,A -85,B 0,C 180,E1 -449.338,E2 -449.338} C_VEL
LIN {X 0,Y 608.434,Z 559,A -85,B 0,C 180,E1 -450,E2 -450} C_VEL
LIN {X 0,Y 608.448,Z 558.184,A -85,B 0,C 180,E1 -451.323,E2 -451.323} C_VEL
LIN {X 0,Y 608.442,Z 557.202,A -85,B 0,C 180,E1 -451.986,E2 -451.986} C_VEL
LIN {X 0,Y 608.425,Z 555.81,A -85,B 0,C 180,E1 -452.648,E2 -452.648} C_VEL
LIN {X 0,Y 608.449,Z 552.897,A -85,B 0,C 180,E1 -453.642,E2 -453.642} C_VEL
LIN {X 0,Y 608.432,Z 548.951,A -85,B 0,C 180,E1 -454.638,E2 -454.638} C_VEL
LIN {X 0,Y 608.437,Z 542.878,A -85,B 0,C 180,E1 -455.801,E2 -455.801} C_VEL
LIN {X 0,Y 608.461,Z 536.237,A -85,B 0,C 180,E1 -456.799,E2 -456.799} C_VEL
LIN {X 0,Y 608.455,Z 527.992,A -85,B 0,C 180,E1 -457.8,E2 -457.8} C_VEL
LIN {X 0,Y 608.477,Z 517.602,A -85,B 0,C 180,E1 -458.803,E2 -458.803} C_VEL
LIN {X 0,Y 608.488,Z 506.752,A -85,B 0,C 180,E1 -459.641,E2 -459.641} C_VEL
LIN {X 0,Y 608.491,Z 495.779,A -85,B 0,C 180,E1 -460.313,E2 -460.313} C_VEL
LIN {X 0,Y 608.534,Z 483.809,A -85,B 0,C 180,E1 -460.888,E2 -460.888} C_VEL
LIN {X 0,Y 608.505,Z 471.889,A -85,B 0,C 180,E1 -461.323,E2 -461.323} C_VEL
LIN {X 0,Y 608.507,Z 459.53,A -85,B 0,C 180,E1 -461.639,E2 -461.639} C_VEL
LIN {X 0,Y 608.531,Z 443.761,A -85,B 0,C 180,E1 -461.871,E2 -461.871} C_VEL
LIN {X 0,Y 608.508,Z 347.172,A -85,B 0,C 180,E1 -463.015,E2 -463.015} C_VEL
LIN {X 0,Y 608.454,Z 346.13,A -85,B 0,C 180,E1 -463.101,E2 -463.101} C_VEL
LIN {X 0,Y 608.467,Z 327.36,A -85,B 0,C 180,E1 -465.577,E2 -465.577} C_VEL
LIN {X 0,Y 608.508,Z 307.944,A -85,B 0,C 180,E1 -468.17,E2 -468.17} C_VEL
LIN {X 0,Y 608.553,Z 287.232,A -85,B 0,C 180,E1 -470.978,E2 -470.978} C_VEL
LIN {X 0,Y 608.461,Z 274.688,A -85,B 0,C 180,E1 -472.714,E2 -472.714} C_VEL
LIN {X 0,Y 608.442,Z 274.689,A -85,B 0,C 180,E1 -475.301,E2 -475.301} C_VEL
LIN {X 0,Y 608.445,Z 274.69,A -85,B 0,C 180,E1 -477.518,E2 -477.518} C_VEL
LIN {X 0,Y 608.464,Z 274.694,A -85,B 0,C 180,E1 -479.97,E2 -479.97} C_VEL
LIN {X 0,Y 608.453,Z 274.687,A -85,B 0,C 180,E1 -482.879,E2 -482.879} C_VEL
LIN {X 0,Y 608.433,Z 274.689,A -85,B 0,C 180,E1 -485.278,E2 -485.278} C_VEL
LIN {X 0,Y 608.466,Z 274.687,A -85,B 0,C 180,E1 -487.746,E2 -487.746} C_VEL
LIN {X 0,Y 608.446,Z 274.698,A -85,B 0,C 180,E1 -490.328,E2 -490.328} C_VEL
LIN {X 0,Y 608.472,Z 274.684,A -85,B 0,C 180,E1 -493.309,E2 -493.309} C_VEL
LIN {X 0,Y 608.462,Z 274.689,A -85,B 0,C 180,E1 -496.13,E2 -496.13} C_VEL
LIN {X 0,Y 608.451,Z 274.694,A -85,B 0,C 180,E1 -498.823,E2 -498.823} C_VEL
LIN {X 0,Y 608.465,Z 274.685,A -85,B 0,C 180,E1 -501.759,E2 -501.759} C_VEL
LIN {X 0,Y 608.457,Z 274.686,A -85,B 0,C 180,E1 -503.952,E2 -503.952} C_VEL
LIN {X 0,Y 608.461,Z 274.689,A -85,B 0,C 180,E1 -506.329,E2 -506.329} C_VEL
LIN {X 0,Y 608.475,Z 274.692,A -85,B 0,C 180,E1 -508.727,E2 -508.727} C_VEL
LIN {X 0,Y 608.46,Z 274.689,A -85,B 0,C 180,E1 -511.381,E2 -511.381} C_VEL
LIN {X 0,Y 608.44,Z 274.688,A -85,B 0,C 180,E1 -513.964,E2 -513.964} C_VEL
LIN {X 0,Y 608.461,Z 274.685,A -85,B 0,C 180,E1 -516.155,E2 -516.155} C_VEL
LIN {X 0,Y 608.455,Z 274.695,A -85,B 0,C 180,E1 -519.018,E2 -519.018} C_VEL
LIN {X 0,Y 608.437,Z 274.69,A -85,B 0,C 180,E1 -521.828,E2 -521.828} C_VEL
LIN {X 0,Y 608.466,Z 274.686,A -85,B 0,C 180,E1 -524.594,E2 -524.594} C_VEL
LIN {X 0,Y 608.476,Z 274.694,A -85,B 0,C 180,E1 -527.323,E2 -527.323} C_VEL
LIN {X 0,Y 608.439,Z 274.69,A -85,B 0,C 180,E1 -530.022,E2 -530.022} C_VEL
LIN {X 0,Y 608.46,Z 274.686,A -85,B 0,C 180,E1 -532.7,E2 -532.7} C_VEL
LIN {X 0,Y 608.456,Z 274.693,A -85,B 0,C 180,E1 -535.362,E2 -535.362} C_VEL
LIN {X 0,Y 608.439,Z 274.693,A -85,B 0,C 180,E1 -538.014,E2 -538.014} C_VEL
LIN {X 0,Y 608.46,Z 274.685,A -85,B 0,C 180,E1 -540.662,E2 -540.662} C_VEL
LIN {X 0,Y 608.483,Z 274.685,A -85,B 0,C 180,E1 -543.311,E2 -543.311} C_VEL
LIN {X 0,Y 608.467,Z 274.695,A -85,B 0,C 180,E1 -545.967,E2 -545.967} C_VEL
LIN {X 0,Y 608.434,Z 274.69,A -85,B 0,C 180,E1 -548.636,E2 -548.636} C_VEL
LIN {X 0,Y 608.461,Z 274.688,A -85,B 0,C 180,E1 -549.441,E2 -549.441} C_VEL
LIN {X 0,Y 607.78,Z 274.782,A -85,B 0,C 180,E1 -549.993,E2 -549.993} C_VEL
LIN {X 0,Y 604.927,Z 275.141,A -85,B 0,C 180,E1 -550.89,E2 -550.89} C_VEL
LIN {X 0,Y 602.523,Z 275.439,A -85,B 0,C 180,E1 -551.611,E2 -551.611} C_VEL
LIN {X 0,Y 601.487,Z 275.564,A -85,B 0,C 180,E1 -552.168,E2 -552.168} C_VEL
LIN {X 0,Y 601.399,Z 275.571,A -85,B 0,C 180,E1 -552.356,E2 -552.356} C_VEL
LIN {X 0,Y 601.396,Z 275.566,A -85,B 0,C 180,E1 -554.898,E2 -554.898} C_VEL
LIN {X 0,Y 601.401,Z 275.565,A -85,B 0,C 180,E1 -556.987,E2 -556.987} C_VEL
LIN {X 0,Y 601.399,Z 275.569,A -85,B 0,C 180,E1 -559.81,E2 -559.81} C_VEL
LIN {X 0,Y 601.404,Z 275.57,A -85,B 0,C 180,E1 -562.683,E2 -562.683} C_VEL
LIN {X 0,Y 601.387,Z 275.57,A -85,B 0,C 180,E1 -564.879,E2 -564.879} C_VEL
LIN {X 0,Y 601.383,Z 275.567,A -85,B 0,C 180,E1 -567.358,E2 -567.358} C_VEL
LIN {X 0,Y 601.394,Z 275.566,A -85,B 0,C 180,E1 -569.394,E2 -569.394} C_VEL
LIN {X 0,Y 601.394,Z 275.566,A -85,B 0,C 180,E1 -571.727,E2 -571.727} C_VEL
LIN {X 0,Y 601.417,Z 275.565,A -85,B 0,C 180,E1 -574.119,E2 -574.119} C_VEL
LIN {X 0,Y 601.424,Z 275.563,A -85,B 0,C 180,E1 -577.382,E2 -577.382} C_VEL
LIN {X 0,Y 601.391,Z 275.566,A -85,B 0,C 180,E1 -579.997,E2 -579.997} C_VEL
LIN {X 0,Y 601.409,Z 275.571,A -85,B 0,C 180,E1 -582.67,E2 -582.67} C_VEL
LIN {X 0,Y 601.393,Z 275.569,A -85,B 0,C 180,E1 -585.48,E2 -585.48} C_VEL
LIN {X 0,Y 601.416,Z 275.564,A -85,B 0,C 180,E1 -588.408,E2 -588.408} C_VEL
LIN {X 0,Y 601.399,Z 275.569,A -85,B 0,C 180,E1 -591.533,E2 -591.533} C_VEL
LIN {X 0,Y 601.385,Z 275.569,A -85,B 0,C 180,E1 -593.742,E2 -593.742} C_VEL
LIN {X 0,Y 601.398,Z 275.565,A -85,B 0,C 180,E1 -596.069,E2 -596.069} C_VEL
LIN {X 0,Y 601.409,Z 275.564,A -85,B 0,C 180,E1 -598.547,E2 -598.547} C_VEL
LIN {X 0,Y 601.427,Z 275.573,A -85,B 0,C 180,E1 -601.373,E2 -601.373} C_VEL
LIN {X 0,Y 601.375,Z 275.569,A -85,B 0,C 180,E1 -604.14,E2 -604.14} C_VEL
LIN {X 0,Y 601.37,Z 275.569,A -85,B 0,C 180,E1 -606.588,E2 -606.588} C_VEL
LIN {X 0,Y 601.429,Z 275.57,A -85,B 0,C 180,E1 -609.479,E2 -609.479} C_VEL
LIN {X 0,Y 601.363,Z 275.571,A -85,B 0,C 180,E1 -612.311,E2 -612.311} C_VEL
LIN {X 0,Y 601.375,Z 275.569,A -85,B 0,C 180,E1 -614.408,E2 -614.408} C_VEL
LIN {X 0,Y 601.394,Z 275.567,A -85,B 0,C 180,E1 -617.172,E2 -617.172} C_VEL
LIN {X 0,Y 601.415,Z 275.575,A -85,B 0,C 180,E1 -619.905,E2 -619.905} C_VEL
LIN {X 0,Y 601.403,Z 275.694,A -85,B 0,C 180,E1 -621.262,E2 -621.262} C_VEL
LIN {X 0,Y 601.45,Z 291.287,A -85,B 0,C 180,E1 -623.964,E2 -623.964} C_VEL
LIN {X 0,Y 601.392,Z 305.052,A -85,B 0,C 180,E1 -626.315,E2 -626.315} C_VEL
LIN {X 0,Y 601.421,Z 308.672,A -85,B 0,C 180,E1 -626.892,E2 -626.892} C_VEL
LIN {X 0,Y 601.669,Z 319.659,A -85,B 0,C 180,E1 -627.029,E2 -627.029} C_VEL
LIN {X 0,Y 601.582,Z 414.738,A -85,B 0,C 180,E1 -628.18,E2 -628.18} C_VEL
LIN {X 0,Y 601.575,Z 427.867,A -85,B 0,C 180,E1 -628.473,E2 -628.473} C_VEL
LIN {X 0,Y 601.558,Z 441.005,A -85,B 0,C 180,E1 -628.912,E2 -628.912} C_VEL
LIN {X 0,Y 601.514,Z 452.123,A -85,B 0,C 180,E1 -629.414,E2 -629.414} C_VEL
LIN {X 0,Y 601.467,Z 463.649,A -85,B 0,C 180,E1 -630.084,E2 -630.084} C_VEL
LIN {X 0,Y 601.451,Z 475.055,A -85,B 0,C 180,E1 -630.921,E2 -630.921} C_VEL
LIN {X 0,Y 601.408,Z 483.306,A -85,B 0,C 180,E1 -631.674,E2 -631.674} C_VEL
LIN {X 0,Y 601.402,Z 491.14,A -85,B 0,C 180,E1 -632.512,E2 -632.512} C_VEL
LIN {X 0,Y 601.357,Z 498.724,A -85,B 0,C 180,E1 -633.518,E2 -633.518} C_VEL
LIN {X 0,Y 601.362,Z 505.747,A -85,B 0,C 180,E1 -634.693,E2 -634.693} C_VEL
LIN {X 0,Y 601.358,Z 510.426,A -85,B 0,C 180,E1 -635.701,E2 -635.701} C_VEL
LIN {X 0,Y 601.354,Z 514.009,A -85,B 0,C 180,E1 -636.712,E2 -636.712} C_VEL
LIN {X 0,Y 601.322,Z 515.862,A -85,B 0,C 180,E1 -637.387,E2 -637.387} C_VEL
LIN {X 0,Y 601.332,Z 517.246,A -85,B 0,C 180,E1 -638.062,E2 -638.062} C_VEL
LIN {X 0,Y 601.335,Z 518.813,A -85,B 0,C 180,E1 -639.417,E2 -639.417} C_VEL
LIN {X 0,Y 601.327,Z 518.994,A -85,B 0,C 180,E1 -640.097,E2 -640.097} C_VEL
LIN {X 0,Y 601.334,Z 518.608,A -85,B 0,C 180,E1 -640.968,E2 -640.968} C_VEL
LIN {X 0,Y 601.343,Z 517.05,A -85,B 0,C 180,E1 -642.144,E2 -642.144} C_VEL
LIN {X 0,Y 601.329,Z 515.532,A -85,B 0,C 180,E1 -642.83,E2 -642.83} C_VEL
LIN {X 0,Y 601.349,Z 511.683,A -85,B 0,C 180,E1 -644.064,E2 -644.064} C_VEL
LIN {X 0,Y 601.356,Z 506.539,A -85,B 0,C 180,E1 -645.246,E2 -645.246} C_VEL
LIN {X 0,Y 601.362,Z 500.603,A -85,B 0,C 180,E1 -646.289,E2 -646.289} C_VEL
LIN {X 0,Y 601.398,Z 493.083,A -85,B 0,C 180,E1 -647.337,E2 -647.337} C_VEL
LIN {X 0,Y 601.421,Z 485.314,A -85,B 0,C 180,E1 -648.216,E2 -648.216} C_VEL
LIN {X 0,Y 601.444,Z 475.921,A -85,B 0,C 180,E1 -649.098,E2 -649.098} C_VEL
LIN {X 0,Y 601.461,Z 465.297,A -85,B 0,C 180,E1 -649.897,E2 -649.897} C_VEL
LIN {X 0,Y 601.507,Z 453.559,A -85,B 0,C 180,E1 -650.599,E2 -650.599} C_VEL
LIN {X 0,Y 601.541,Z 441.379,A -85,B 0,C 180,E1 -651.164,E2 -651.164} C_VEL
LIN {X 0,Y 601.509,Z 428.692,A -85,B 0,C 180,E1 -651.595,E2 -651.595} C_VEL
LIN {X 0,Y 601.533,Z 416.018,A -85,B 0,C 180,E1 -651.887,E2 -651.887} C_VEL
LIN {X 0,Y 601.574,Z 369.749,A -85,B 0,C 180,E1 -652.463,E2 -652.463} C_VEL
LIN {X 0,Y 601.599,Z 309.686,A -85,B 0,C 180,E1 -653.182,E2 -653.182} C_VEL
LIN {X 0,Y 601.396,Z 308.265,A -85,B 0,C 180,E1 -653.229,E2 -653.229} C_VEL
LIN {X 0,Y 601.411,Z 292.804,A -85,B 0,C 180,E1 -655.867,E2 -655.867} C_VEL
LIN {X 0,Y 601.489,Z 276.847,A -85,B 0,C 180,E1 -658.624,E2 -658.624} C_VEL
LIN {X 0,Y 601.453,Z 275.561,A -85,B 0,C 180,E1 -658.89,E2 -658.89} C_VEL
LIN {X 0,Y 601.4,Z 275.568,A -85,B 0,C 180,E1 -661.727,E2 -661.727} C_VEL
LIN {X 0,Y 601.418,Z 275.571,A -85,B 0,C 180,E1 -664.119,E2 -664.119} C_VEL
LIN {X 0,Y 601.435,Z 275.56,A -85,B 0,C 180,E1 -667.382,E2 -667.382} C_VEL
LIN {X 0,Y 601.399,Z 275.568,A -85,B 0,C 180,E1 -669.996,E2 -669.996} C_VEL
LIN {X 0,Y 601.409,Z 275.574,A -85,B 0,C 180,E1 -672.67,E2 -672.67} C_VEL
LIN {X 0,Y 601.397,Z 275.566,A -85,B 0,C 180,E1 -675.479,E2 -675.479} C_VEL
LIN {X 0,Y 601.42,Z 275.568,A -85,B 0,C 180,E1 -678.407,E2 -678.407} C_VEL
LIN {X 0,Y 601.432,Z 275.562,A -85,B 0,C 180,E1 -681.529,E2 -681.529} C_VEL
LIN {X 0,Y 601.383,Z 275.568,A -85,B 0,C 180,E1 -684.245,E2 -684.245} C_VEL
LIN {X 0,Y 601.413,Z 275.569,A -85,B 0,C 180,E1 -686.686,E2 -686.686} C_VEL
LIN {X 0,Y 601.414,Z 275.574,A -85,B 0,C 180,E1 -689.058,E2 -689.058} C_VEL
LIN {X 0,Y 601.431,Z 275.568,A -85,B 0,C 180,E1 -691.373,E2 -691.373} C_VEL
LIN {X 0,Y 601.41,Z 275.564,A -85,B 0,C 180,E1 -694.133,E2 -694.133} C_VEL
LIN {X 0,Y 601.417,Z 275.563,A -85,B 0,C 180,E1 -696.59,E2 -696.59} C_VEL
LIN {X 0,Y 601.43,Z 275.571,A -85,B 0,C 180,E1 -699.478,E2 -699.478} C_VEL
LIN {X 0,Y 601.39,Z 275.566,A -85,B 0,C 180,E1 -702.312,E2 -702.312} C_VEL
LIN {X 0,Y 601.409,Z 275.564,A -85,B 0,C 180,E1 -704.409,E2 -704.409} C_VEL
LIN {X 0,Y 601.414,Z 275.567,A -85,B 0,C 180,E1 -707.172,E2 -707.172} C_VEL
LIN {X 0,Y 601.427,Z 275.57,A -85,B 0,C 180,E1 -709.905,E2 -709.905} C_VEL
LIN {X 0,Y 601.439,Z 275.56,A -85,B 0,C 180,E1 -712.615,E2 -712.615} C_VEL
LIN {X 0,Y 601.412,Z 275.565,A -85,B 0,C 180,E1 -715.308,E2 -715.308} C_VEL
LIN {X 0,Y 601.432,Z 275.572,A -85,B 0,C 180,E1 -717.991,E2 -717.991} C_VEL
LIN {X 0,Y 601.443,Z 275.561,A -85,B 0,C 180,E1 -720.67,E2 -720.67} C_VEL
LIN {X 0,Y 601.43,Z 275.561,A -85,B 0,C 180,E1 -723.35,E2 -723.35} C_VEL
LIN {X 0,Y 601.404,Z 275.572,A -85,B 0,C 180,E1 -726.037,E2 -726.037} C_VEL
LIN {X 0,Y 601.415,Z 275.567,A -85,B 0,C 180,E1 -728.738,E2 -728.738} C_VEL
LIN {X 0,Y 601.432,Z 275.561,A -85,B 0,C 180,E1 -731.458,E2 -731.458} C_VEL
LIN {X 0,Y 601.419,Z 275.569,A -85,B 0,C 180,E1 -734.206,E2 -734.206} C_VEL
LIN {X 0,Y 601.429,Z 275.565,A -85,B 0,C 180,E1 -736.986,E2 -736.986} C_VEL
LIN {X 0,Y 601.401,Z 275.565,A -85,B 0,C 180,E1 -739.81,E2 -739.81} C_VEL
LIN {X 0,Y 601.415,Z 275.572,A -85,B 0,C 180,E1 -742.606,E2 -742.606} C_VEL
LIN {X 0,Y 601.398,Z 275.575,A -85,B 0,C 180,E1 -744.879,E2 -744.879} C_VEL
LIN {X 0,Y 601.413,Z 275.566,A -85,B 0,C 180,E1 -747.362,E2 -747.362} C_VEL
LIN {X 0,Y 601.429,Z 275.562,A -85,B 0,C 180,E1 -750.164,E2 -750.164} C_VEL
LIN {X 0,Y 601.417,Z 275.568,A -85,B 0,C 180,E1 -752.715,E2 -752.715} C_VEL
LIN {X 0,Y 601.392,Z 275.578,A -85,B 0,C 180,E1 -755.112,E2 -755.112} C_VEL
LIN {X 0,Y 601.436,Z 275.568,A -85,B 0,C 180,E1 -757.419,E2 -757.419} C_VEL
LIN {X 0,Y 601.401,Z 275.565,A -85,B 0,C 180,E1 -759.996,E2 -759.996} C_VEL
LIN {X 0,Y 601.413,Z 275.564,A -85,B 0,C 180,E1 -762.67,E2 -762.67} C_VEL
LIN {X 0,Y 601.399,Z 275.576,A -85,B 0,C 180,E1 -765.48,E2 -765.48} C_VEL
LIN {X 0,Y 601.423,Z 275.562,A -85,B 0,C 180,E1 -768.407,E2 -768.407} C_VEL
LIN {X 0,Y 601.428,Z 275.571,A -85,B 0,C 180,E1 -771.53,E2 -771.53} C_VEL
LIN {X 0,Y 601.384,Z 275.57,A -85,B 0,C 180,E1 -774.245,E2 -774.245} C_VEL
LIN {X 0,Y 601.416,Z 275.563,A -85,B 0,C 180,E1 -776.686,E2 -776.686} C_VEL
LIN {X 0,Y 601.416,Z 275.564,A -85,B 0,C 180,E1 -779.058,E2 -779.058} C_VEL
LIN {X 0,Y 601.43,Z 275.564,A -85,B 0,C 180,E1 -781.373,E2 -781.373} C_VEL
LIN {X 0,Y 601.399,Z 275.57,A -85,B 0,C 180,E1 -783.636,E2 -783.636} C_VEL
LIN {X 0,Y 601.418,Z 275.569,A -85,B 0,C 180,E1 -786.59,E2 -786.59} C_VEL
LIN {X 0,Y 601.421,Z 275.578,A -85,B 0,C 180,E1 -787.136,E2 -787.136} C_VEL
LIN {X 0,Y 601.673,Z 282.051,A -85,B 0,C 180,E1 -788.051,E2 -788.051} C_VEL
LIN {X 0,Y 601.602,Z 302.762,A -85,B 0,C 180,E1 -790.907,E2 -790.907} C_VEL
LIN {X 0,Y 601.524,Z 323.473,A -85,B 0,C 180,E1 -793.715,E2 -793.715} C_VEL
LIN {X 0,Y 601.468,Z 344.185,A -85,B 0,C 180,E1 -796.485,E2 -796.485} C_VEL
LIN {X 0,Y 601.426,Z 346.612,A -85,B 0,C 180,E1 -796.807,E2 -796.807} C_VEL
LIN {X 0,Y 601.667,Z 350.709,A -85,B 0,C 180,E1 -796.877,E2 -796.877} C_VEL
LIN {X 0,Y 601.594,Z 454.939,A -85,B 0,C 180,E1 -798.139,E2 -798.139} C_VEL
LIN {X 0,Y 601.556,Z 468.212,A -85,B 0,C 180,E1 -798.437,E2 -798.437} C_VEL
LIN {X 0,Y 601.542,Z 479.915,A -85,B 0,C 180,E1 -798.826,E2 -798.826} C_VEL
LIN {X 0,Y 601.521,Z 492.631,A -85,B 0,C 180,E1 -799.396,E2 -799.396} C_VEL
LIN {X 0,Y 601.472,Z 504.196,A -85,B 0,C 180,E1 -800.075,E2 -800.075} C_VEL
LIN {X 0,Y 601.444,Z 514.593,A -85,B 0,C 180,E1 -800.839,E2 -800.839} C_VEL
LIN {X 0,Y 601.405,Z 523.014,A -85,B 0,C 180,E1 -801.6,E2 -801.6} C_VEL
LIN {X 0,Y 601.418,Z 530.959,A -85,B 0,C 180,E1 -802.446,E2 -802.446} C_VEL
LIN {X 0,Y 601.366,Z 538.248,A -85,B 0,C 180,E1 -803.401,E2 -803.401} C_VEL
LIN {X 0,Y 601.372,Z 543.865,A -85,B 0,C 180,E1 -804.299,E2 -804.299} C_VEL
LIN {X 0,Y 601.336,Z 548.949,A -85,B 0,C 180,E1 -805.307,E2 -805.307} C_VEL
LIN {X 0,Y 601.367,Z 552.895,A -85,B 0,C 180,E1 -806.314,E2 -806.314} C_VEL
LIN {X 0,Y 601.325,Z 555.808,A -85,B 0,C 180,E1 -807.32,E2 -807.32} C_VEL
LIN {X 0,Y 601.341,Z 557.201,A -85,B 0,C 180,E1 -807.99,E2 -807.99} C_VEL
LIN {X 0,Y 601.339,Z 558.784,A -85,B 0,C 180,E1 -809.33,E2 -809.33} C_VEL
LIN {X 0,Y 601.335,Z 559,A -85,B 0,C 180,E1 -810,E2 -810} C_VEL
LIN {X 0,Y 601.347,Z 558.185,A -85,B 0,C 180,E1 -811.339,E2 -811.339} C_VEL
LIN {X 0,Y 601.341,Z 557.202,A -85,B 0,C 180,E1 -812.009,E2 -812.009} C_VEL
LIN {X 0,Y 601.325,Z 555.81,A -85,B 0,C 180,E1 -812.679,E2 -812.679} C_VEL
LIN {X 0,Y 601.367,Z 552.897,A -85,B 0,C 180,E1 -813.685,E2 -813.685} C_VEL
LIN {X 0,Y 601.336,Z 548.951,A -85,B 0,C 180,E1 -814.692,E2 -814.692} C_VEL
LIN {X 0,Y 601.372,Z 542.879,A -85,B 0,C 180,E1 -815.869,E2 -815.869} C_VEL
LIN {X 0,Y 601.381,Z 536.238,A -85,B 0,C 180,E1 -816.879,E2 -816.879} C_VEL
LIN {X 0,Y 601.4,Z 527.992,A -85,B 0,C 180,E1 -817.892,E2 -817.892} C_VEL
LIN {X 0,Y 601.434,Z 517.603,A -85,B 0,C 180,E1 -818.907,E2 -818.907} C_VEL
LIN {X 0,Y 601.46,Z 506.752,A -85,B 0,C 180,E1 -819.754,E2 -819.754} C_VEL
LIN {X 0,Y 601.494,Z 495.781,A -85,B 0,C 180,E1 -820.434,E2 -820.434} C_VEL
LIN {X 0,Y 601.548,Z 483.683,A -85,B 0,C 180,E1 -821.022,E2 -821.022} C_VEL
LIN {X 0,Y 601.53,Z 471.888,A -85,B 0,C 180,E1 -821.456,E2 -821.456} C_VEL
LIN {X 0,Y 601.577,Z 459.529,A -85,B 0,C 180,E1 -821.775,E2 -821.775} C_VEL
LIN {X 0,Y 601.607,Z 443.761,A -85,B 0,C 180,E1 -822.01,E2 -822.01} C_VEL
LIN {X 0,Y 601.479,Z 347.172,A -85,B 0,C 180,E1 -823.17,E2 -823.17} C_VEL
LIN {X 0,Y 601.461,Z 346.13,A -85,B 0,C 180,E1 -823.256,E2 -823.256} C_VEL
LIN {X 0,Y 601.466,Z 326.066,A -85,B 0,C 180,E1 -825.937,E2 -825.937} C_VEL
LIN {X 0,Y 601.574,Z 306.211,A -85,B 0,C 180,E1 -828.623,E2 -828.623} C_VEL
LIN {X 0,Y 601.654,Z 284.643,A -85,B 0,C 180,E1 -831.589,E2 -831.589} C_VEL
LIN {X 0,Y 601.673,Z 276.877,A -85,B 0,C 180,E1 -832.672,E2 -832.672} C_VEL
LIN {X 0,Y 601.417,Z 275.567,A -85,B 0,C 180,E1 -832.887,E2 -832.887} C_VEL
LIN {X 0,Y 601.398,Z 275.566,A -85,B 0,C 180,E1 -834.878,E2 -834.878} C_VEL
LIN {X 0,Y 601.413,Z 275.565,A -85,B 0,C 180,E1 -837.361,E2 -837.361} C_VEL
LIN {X 0,Y 601.429,Z 275.572,A -85,B 0,C 180,E1 -840.163,E2 -840.163} C_VEL
LIN {X 0,Y 601.419,Z 275.565,A -85,B 0,C 180,E1 -842.714,E2 -842.714} C_VEL
LIN {X 0,Y 601.39,Z 275.566,A -85,B 0,C 180,E1 -845.111,E2 -845.111} C_VEL
LIN {X 0,Y 601.434,Z 275.561,A -85,B 0,C 180,E1 -847.418,E2 -847.418} C_VEL
LIN {X 0,Y 601.399,Z 275.57,A -85,B 0,C 180,E1 -849.995,E2 -849.995} C_VEL
LIN {X 0,Y 601.41,Z 275.571,A -85,B 0,C 180,E1 -852.67,E2 -852.67} C_VEL
LIN {X 0,Y 601.396,Z 275.565,A -85,B 0,C 180,E1 -855.479,E2 -855.479} C_VEL
LIN {X 0,Y 601.423,Z 275.57,A -85,B 0,C 180,E1 -858.406,E2 -858.406} C_VEL
LIN {X 0,Y 601.429,Z 275.562,A -85,B 0,C 180,E1 -861.528,E2 -861.528} C_VEL
LIN {X 0,Y 601.391,Z 275.569,A -85,B 0,C 180,E1 -864.245,E2 -864.245} C_VEL
LIN {X 0,Y 601.423,Z 275.571,A -85,B 0,C 180,E1 -866.686,E2 -866.686} C_VEL
LIN {X 0,Y 601.428,Z 275.57,A -85,B 0,C 180,E1 -869.058,E2 -869.058} C_VEL
LIN {X 0,Y 601.42,Z 275.566,A -85,B 0,C 180,E1 -871.372,E2 -871.372} C_VEL
LIN {X 0,Y 601.399,Z 275.567,A -85,B 0,C 180,E1 -873.636,E2 -873.636} C_VEL
LIN {X 0,Y 601.417,Z 275.566,A -85,B 0,C 180,E1 -876.589,E2 -876.589} C_VEL
LIN {X 0,Y 601.423,Z 275.568,A -85,B 0,C 180,E1 -879.478,E2 -879.478} C_VEL
LIN {X 0,Y 601.389,Z 275.566,A -85,B 0,C 180,E1 -882.311,E2 -882.311} C_VEL
LIN {X 0,Y 601.407,Z 275.564,A -85,B 0,C 180,E1 -884.408,E2 -884.408} C_VEL
LIN {X 0,Y 601.42,Z 275.57,A -85,B 0,C 180,E1 -887.172,E2 -887.172} C_VEL
LIN {X 0,Y 601.42,Z 275.566,A -85,B 0,C 180,E1 -889.905,E2 -889.905} C_VEL
LIN {X 0,Y 601.435,Z 275.561,A -85,B 0,C 180,E1 -892.615,E2 -892.615} C_VEL
LIN {X 0,Y 601.424,Z 275.568,A -85,B 0,C 180,E1 -895.308,E2 -895.308} C_VEL
LIN {X 0,Y 601.41,Z 275.569,A -85,B 0,C 180,E1 -897.991,E2 -897.991} C_VEL
LIN {X 0,Y 601.433,Z 275.561,A -85,B 0,C 180,E1 -900.669,E2 -900.669} C_VEL
LIN {X 0,Y 601.434,Z 275.564,A -85,B 0,C 180,E1 -903.349,E2 -903.349} C_VEL
LIN {X 0,Y 601.415,Z 275.572,A -85,B 0,C 180,E1 -906.037,E2 -906.037} C_VEL
LIN {X 0,Y 601.435,Z 275.57,A -85,B 0,C 180,E1 -908.061,E2 -908.061} C_VEL
LIN {X 0,Y 601.408,Z 275.564,A -85,B 0,C 180,E1 -911.007,E2 -911.007} C_VEL
LIN {X 0,Y 601.399,Z 275.571,A -85,B 0,C 180,E1 -912.356,E2 -912.356} C_VEL
LIN {X 0,Y 600.724,Z 275.651,A -85,B 0,C 180,E1 -912.916,E2 -912.916} C_VEL
LIN {X 0,Y 597.864,Z 276.012,A -85,B 0,C 180,E1 -913.824,E2 -913.824} C_VEL
LIN {X 0,Y 595.456,Z 276.309,A -85,B 0,C 180,E1 -914.554,E2 -914.554} C_VEL
LIN {X 0,Y 594.425,Z 276.434,A -85,B 0,C 180,E1 -915.117,E2 -915.117} C_VEL
LIN {X 0,Y 594.343,Z 276.444,A -85,B 0,C 180,E1 -915.308,E2 -915.308} C_VEL
LIN {X 0,Y 594.345,Z 276.449,A -85,B 0,C 180,E1 -917.905,E2 -917.905} C_VEL
LIN {X 0,Y 594.39,Z 276.441,A -85,B 0,C 180,E1 -920.776,E2 -920.776} C_VEL
LIN {X 0,Y 594.373,Z 276.442,A -85,B 0,C 180,E1 -923.705,E2 -923.705} C_VEL
LIN {X 0,Y 594.363,Z 276.448,A -85,B 0,C 180,E1 -926.7,E2 -926.7} C_VEL
LIN {X 0,Y 594.371,Z 276.444,A -85,B 0,C 180,E1 -928.999,E2 -928.999} C_VEL
LIN {X 0,Y 594.368,Z 276.441,A -85,B 0,C 180,E1 -931.642,E2 -931.642} C_VEL
LIN {X 0,Y 594.372,Z 276.45,A -85,B 0,C 180,E1 -934.58,E2 -934.58} C_VEL
LIN {X 0,Y 594.38,Z 276.44,A -85,B 0,C 180,E1 -937.608,E2 -937.608} C_VEL
LIN {X 0,Y 594.361,Z 276.448,A -85,B 0,C 180,E1 -940.568,E2 -940.568} C_VEL
LIN {X 0,Y 594.347,Z 276.448,A -85,B 0,C 180,E1 -943.301,E2 -943.301} C_VEL
LIN {X 0,Y 594.355,Z 276.443,A -85,B 0,C 180,E1 -946.162,E2 -946.162} C_VEL
LIN {X 0,Y 594.372,Z 276.45,A -85,B 0,C 180,E1 -949.178,E2 -949.178} C_VEL
LIN {X 0,Y 594.366,Z 276.441,A -85,B 0,C 180,E1 -952.058,E2 -952.058} C_VEL
LIN {X 0,Y 594.348,Z 276.446,A -85,B 0,C 180,E1 -954.677,E2 -954.677} C_VEL
LIN {X 0,Y 594.372,Z 276.448,A -85,B 0,C 180,E1 -957.089,E2 -957.089} C_VEL
LIN {X 0,Y 594.345,Z 276.449,A -85,B 0,C 180,E1 -959.679,E2 -959.679} C_VEL
LIN {X 0,Y 594.357,Z 276.447,A -85,B 0,C 180,E1 -961.773,E2 -961.773} C_VEL
LIN {X 0,Y 594.335,Z 276.447,A -85,B 0,C 180,E1 -964.055,E2 -964.055} C_VEL
LIN {X 0,Y 594.352,Z 276.444,A -85,B 0,C 180,E1 -966.295,E2 -966.295} C_VEL
LIN {X 0,Y 594.404,Z 276.441,A -85,B 0,C 180,E1 -969.225,E2 -969.225} C_VEL
LIN {X 0,Y 594.33,Z 276.45,A -85,B 0,C 180,E1 -972.095,E2 -972.095} C_VEL
LIN {X 0,Y 594.336,Z 276.448,A -85,B 0,C 180,E1 -974.219,E2 -974.219} C_VEL
LIN {X 0,Y 594.346,Z 276.447,A -85,B 0,C 180,E1 -976.321,E2 -976.321} C_VEL
LIN {X 0,Y 594.329,Z 276.447,A -85,B 0,C 180,E1 -978.956,E2 -978.956} C_VEL
LIN {X 0,Y 594.366,Z 276.531,A -85,B 0,C 180,E1 -981.179,E2 -981.179} C_VEL
LIN {X 0,Y 594.412,Z 288.088,A -85,B 0,C 180,E1 -983.21,E2 -983.21} C_VEL
LIN {X 0,Y 594.352,Z 303.79,A -85,B 0,C 180,E1 -985.932,E2 -985.932} C_VEL
LIN {X 0,Y 594.342,Z 308.353,A -85,B 0,C 180,E1 -986.717,E2 -986.717} C_VEL
LIN {X 0,Y 594.756,Z 312.05,A -85,B 0,C 180,E1 -986.783,E2 -986.783} C_VEL
LIN {X 0,Y 594.631,Z 415.461,A -85,B 0,C 180,E1 -988.053,E2 -988.053} C_VEL
LIN {X 0,Y 594.631,Z 429.08,A -85,B 0,C 180,E1 -988.371,E2 -988.371} C_VEL
LIN {X 0,Y 594.595,Z 441.887,A -85,B 0,C 180,E1 -988.815,E2 -988.815} C_VEL
LIN {X 0,Y 594.52,Z 452.783,A -85,B 0,C 180,E1 -989.323,E2 -989.323} C_VEL
LIN {X 0,Y 594.452,Z 464.172,A -85,B 0,C 180,E1 -990,E2 -990} C_VEL
LIN {X 0,Y 594.424,Z 474.443,A -85,B 0,C 180,E1 -990.762,E2 -990.762} C_VEL
LIN {X 0,Y 594.361,Z 482.828,A -85,B 0,C 180,E1 -991.525,E2 -991.525} C_VEL
LIN {X 0,Y 594.332,Z 490.721,A -85,B 0,C 180,E1 -992.372,E2 -992.372} C_VEL
LIN {X 0,Y 594.276,Z 498.398,A -85,B 0,C 180,E1 -993.39,E2 -993.39} C_VEL
LIN {X 0,Y 594.277,Z 504.576,A -85,B 0,C 180,E1 -994.409,E2 -994.409} C_VEL
LIN {X 0,Y 594.27,Z 509.505,A -85,B 0,C 180,E1 -995.429,E2 -995.429} C_VEL
LIN {X 0,Y 594.267,Z 513.728,A -85,B 0,C 180,E1 -996.581,E2 -996.581} C_VEL
LIN {X 0,Y 594.247,Z 516.123,A -85,B 0,C 180,E1 -997.475,E2 -997.475} C_VEL
LIN {X 0,Y 594.228,Z 517.442,A -85,B 0,C 180,E1 -998.159,E2 -998.159} C_VEL
LIN {X 0,Y 594.227,Z 518.363,A -85,B 0,C 180,E1 -998.845,E2 -998.845} C_VEL
LIN {X 0,Y 594.255,Z 518.885,A -85,B 0,C 180,E1 -999.531,E2 -999.531} C_VEL
LIN {X 0,Y 594.237,Z 518.657,A -85,B 0,C 180,E1 -1000.908,E2 -1000.908} C_VEL
LIN {X 0,Y 594.232,Z 517.953,A -85,B 0,C 180,E1 -1001.599,E2 -1001.599} C_VEL
LIN {X 0,Y 594.24,Z 516.806,A -85,B 0,C 180,E1 -1002.292,E2 -1002.292} C_VEL
LIN {X 0,Y 594.256,Z 514.273,A -85,B 0,C 180,E1 -1003.334,E2 -1003.334} C_VEL
LIN {X 0,Y 594.256,Z 510.678,A -85,B 0,C 180,E1 -1004.38,E2 -1004.38} C_VEL
LIN {X 0,Y 594.266,Z 505.903,A -85,B 0,C 180,E1 -1005.432,E2 -1005.432} C_VEL
LIN {X 0,Y 594.314,Z 499.789,A -85,B 0,C 180,E1 -1006.488,E2 -1006.488} C_VEL
LIN {X 0,Y 594.331,Z 492.084,A -85,B 0,C 180,E1 -1007.55,E2 -1007.55} C_VEL
LIN {X 0,Y 594.386,Z 484.078,A -85,B 0,C 180,E1 -1008.439,E2 -1008.439} C_VEL
LIN {X 0,Y 594.397,Z 476.006,A -85,B 0,C 180,E1 -1009.199,E2 -1009.199} C_VEL
LIN {X 0,Y 594.452,Z 466.085,A -85,B 0,C 180,E1 -1009.961,E2 -1009.961} C_VEL
LIN {X 0,Y 594.512,Z 454.358,A -85,B 0,C 180,E1 -1010.681,E2 -1010.681} C_VEL
LIN {X 0,Y 594.568,Z 441.885,A -85,B 0,C 180,E1 -1011.276,E2 -1011.276} C_VEL
LIN {X 0,Y 594.561,Z 429.787,A -85,B 0,C 180,E1 -1011.701,E2 -1011.701} C_VEL
LIN {X 0,Y 594.58,Z 416.447,A -85,B 0,C 180,E1 -1012.019,E2 -1012.019} C_VEL
LIN {X 0,Y 594.638,Z 387.713,A -85,B 0,C 180,E1 -1012.392,E2 -1012.392} C_VEL
LIN {X 0,Y 594.596,Z 309.981,A -85,B 0,C 180,E1 -1013.336,E2 -1013.336} C_VEL
LIN {X 0,Y 594.358,Z 308.3,A -85,B 0,C 180,E1 -1013.382,E2 -1013.382} C_VEL
LIN {X 0,Y 594.444,Z 291.288,A -85,B 0,C 180,E1 -1016.321,E2 -1016.321} C_VEL
LIN {X 0,Y 594.426,Z 276.457,A -85,B 0,C 180,E1 -1018.922,E2 -1018.922} C_VEL
LIN {X 0,Y 594.376,Z 276.443,A -85,B 0,C 180,E1 -1021.642,E2 -1021.642} C_VEL
LIN {X 0,Y 594.376,Z 276.447,A -85,B 0,C 180,E1 -1024.58,E2 -1024.58} C_VEL
LIN {X 0,Y 594.388,Z 276.438,A -85,B 0,C 180,E1 -1027.608,E2 -1027.608} C_VEL
LIN {X 0,Y 594.367,Z 276.452,A -85,B 0,C 180,E1 -1030.567,E2 -1030.567} C_VEL
LIN {X 0,Y 594.365,Z 276.442,A -85,B 0,C 180,E1 -1033.299,E2 -1033.299} C_VEL
LIN {X 0,Y 594.359,Z 276.445,A -85,B 0,C 180,E1 -1036.161,E2 -1036.161} C_VEL
LIN {X 0,Y 594.378,Z 276.447,A -85,B 0,C 180,E1 -1038.536,E2 -1038.536} C_VEL
LIN {X 0,Y 594.382,Z 276.443,A -85,B 0,C 180,E1 -1041.296,E2 -1041.296} C_VEL
LIN {X 0,Y 594.351,Z 276.443,A -85,B 0,C 180,E1 -1043.756,E2 -1043.756} C_VEL
LIN {X 0,Y 594.374,Z 276.441,A -85,B 0,C 180,E1 -1046.239,E2 -1046.239} C_VEL
LIN {X 0,Y 594.368,Z 276.445,A -85,B 0,C 180,E1 -1048.65,E2 -1048.65} C_VEL
LIN {X 0,Y 594.382,Z 276.448,A -85,B 0,C 180,E1 -1051.042,E2 -1051.042} C_VEL
LIN {X 0,Y 594.384,Z 276.439,A -85,B 0,C 180,E1 -1053.977,E2 -1053.977} C_VEL
LIN {X 0,Y 594.387,Z 276.438,A -85,B 0,C 180,E1 -1056.296,E2 -1056.296} C_VEL
LIN {X 0,Y 594.403,Z 276.445,A -85,B 0,C 180,E1 -1059.225,E2 -1059.225} C_VEL
LIN {X 0,Y 594.35,Z 276.445,A -85,B 0,C 180,E1 -1062.095,E2 -1062.095} C_VEL
LIN {X 0,Y 594.363,Z 276.442,A -85,B 0,C 180,E1 -1064.219,E2 -1064.219} C_VEL
LIN {X 0,Y 594.379,Z 276.441,A -85,B 0,C 180,E1 -1066.321,E2 -1066.321} C_VEL
LIN {X 0,Y 594.37,Z 276.442,A -85,B 0,C 180,E1 -1069.095,E2 -1069.095} C_VEL
LIN {X 0,Y 594.409,Z 276.446,A -85,B 0,C 180,E1 -1071.843,E2 -1071.843} C_VEL
LIN {X 0,Y 594.393,Z 276.439,A -85,B 0,C 180,E1 -1074.572,E2 -1074.572} C_VEL
LIN {X 0,Y 594.4,Z 276.438,A -85,B 0,C 180,E1 -1077.289,E2 -1077.289} C_VEL
LIN {X 0,Y 594.413,Z 276.446,A -85,B 0,C 180,E1 -1080,E2 -1080} C_VEL
LIN {X 0,Y 594.402,Z 276.438,A -85,B 0,C 180,E1 -1082.711,E2 -1082.711} C_VEL
LIN {X 0,Y 594.392,Z 276.438,A -85,B 0,C 180,E1 -1085.428,E2 -1085.428} C_VEL
LIN {X 0,Y 594.408,Z 276.444,A -85,B 0,C 180,E1 -1088.157,E2 -1088.157} C_VEL
LIN {X 0,Y 594.388,Z 276.439,A -85,B 0,C 180,E1 -1091.074,E2 -1091.074} C_VEL
LIN {X 0,Y 594.38,Z 276.44,A -85,B 0,C 180,E1 -1093.679,E2 -1093.679} C_VEL
LIN {X 0,Y 594.393,Z 276.446,A -85,B 0,C 180,E1 -1096.719,E2 -1096.719} C_VEL
LIN {X 0,Y 594.366,Z 276.442,A -85,B 0,C 180,E1 -1099.335,E2 -1099.335} C_VEL
LIN {X 0,Y 594.361,Z 276.442,A -85,B 0,C 180,E1 -1101.504,E2 -1101.504} C_VEL
LIN {X 0,Y 594.389,Z 276.443,A -85,B 0,C 180,E1 -1104.446,E2 -1104.446} C_VEL
LIN {X 0,Y 594.382,Z 276.448,A -85,B 0,C 180,E1 -1106.7,E2 -1106.7} C_VEL
LIN {X 0,Y 594.38,Z 276.45,A -85,B 0,C 180,E1 -1108.999,E2 -1108.999} C_VEL
LIN {X 0,Y 594.376,Z 276.441,A -85,B 0,C 180,E1 -1111.643,E2 -1111.643} C_VEL
LIN {X 0,Y 594.379,Z 276.442,A -85,B 0,C 180,E1 -1114.58,E2 -1114.58} C_VEL
LIN {X 0,Y 594.39,Z 276.442,A -85,B 0,C 180,E1 -1117.609,E2 -1117.609} C_VEL
LIN {X 0,Y 594.368,Z 276.441,A -85,B 0,C 180,E1 -1120.567,E2 -1120.567} C_VEL
LIN {X 0,Y 594.368,Z 276.451,A -85,B 0,C 180,E1 -1123.3,E2 -1123.3} C_VEL
LIN {X 0,Y 594.361,Z 276.443,A -85,B 0,C 180,E1 -1126.162,E2 -1126.162} C_VEL
LIN {X 0,Y 594.38,Z 276.439,A -85,B 0,C 180,E1 -1128.536,E2 -1128.536} C_VEL
LIN {X 0,Y 594.381,Z 276.445,A -85,B 0,C 180,E1 -1131.297,E2 -1131.297} C_VEL
LIN {X 0,Y 594.352,Z 276.454,A -85,B 0,C 180,E1 -1133.756,E2 -1133.756} C_VEL
LIN {X 0,Y 594.365,Z 276.445,A -85,B 0,C 180,E1 -1136.238,E2 -1136.238} C_VEL
LIN {X 0,Y 594.37,Z 276.441,A -85,B 0,C 180,E1 -1138.65,E2 -1138.65} C_VEL
LIN {X 0,Y 594.384,Z 276.439,A -85,B 0,C 180,E1 -1141.043,E2 -1141.043} C_VEL
LIN {X 0,Y 594.381,Z 276.45,A -85,B 0,C 180,E1 -1143.979,E2 -1143.979} C_VEL
LIN {X 0,Y 594.386,Z 276.446,A -85,B 0,C 180,E1 -1146.665,E2 -1146.665} C_VEL
LIN {X 0,Y 594.403,Z 276.549,A -85,B 0,C 180,E1 -1146.988,E2 -1146.988} C_VEL
LIN {X 0,Y 594.765,Z 281.023,A -85,B 0,C 180,E1 -1147.637,E2 -1147.637} C_VEL
LIN {X 0,Y 594.637,Z 302.762,A -85,B 0,C 180,E1 -1150.675,E2 -1150.675} C_VEL
LIN {X 0,Y 594.554,Z 323.473,A -85,B 0,C 180,E1 -1153.519,E2 -1153.519} C_VEL
LIN {X 0,Y 594.439,Z 345.479,A -85,B 0,C 180,E1 -1156.497,E2 -1156.497} C_VEL
LIN {X 0,Y 594.442,Z 346.612,A -85,B 0,C 180,E1 -1156.649,E2 -1156.649} C_VEL
LIN {X 0,Y 594.776,Z 350.709,A -85,B 0,C 180,E1 -1156.722,E2 -1156.722} C_VEL
LIN {X 0,Y 594.646,Z 454.939,A -85,B 0,C 180,E1 -1157.998,E2 -1157.998} C_VEL
LIN {X 0,Y 594.621,Z 468.213,A -85,B 0,C 180,E1 -1158.301,E2 -1158.301} C_VEL
LIN {X 0,Y 594.574,Z 480.501,A -85,B 0,C 180,E1 -1158.715,E2 -1158.715} C_VEL
LIN {X 0,Y 594.533,Z 492.629,A -85,B 0,C 180,E1 -1159.27,E2 -1159.27} C_VEL
LIN {X 0,Y 594.46,Z 504.198,A -85,B 0,C 180,E1 -1159.957,E2 -1159.957} C_VEL
LIN {X 0,Y 594.413,Z 514.595,A -85,B 0,C 180,E1 -1160.729,E2 -1160.729} C_VEL
LIN {X 0,Y 594.349,Z 523.027,A -85,B 0,C 180,E1 -1161.5,E2 -1161.5} C_VEL
LIN {X 0,Y 594.347,Z 530.959,A -85,B 0,C 180,E1 -1162.355,E2 -1162.355} C_VEL
LIN {X 0,Y 594.281,Z 538.824,A -85,B 0,C 180,E1 -1163.41,E2 -1163.41} C_VEL
LIN {X 0,Y 594.289,Z 545.679,A -85,B 0,C 180,E1 -1164.571,E2 -1164.571} C_VEL
LIN {X 0,Y 594.27,Z 550.37,A -85,B 0,C 180,E1 -1165.591,E2 -1165.591} C_VEL
LIN {X 0,Y 594.267,Z 553.956,A -85,B 0,C 180,E1 -1166.61,E2 -1166.61} C_VEL
LIN {X 0,Y 594.226,Z 555.808,A -85,B 0,C 180,E1 -1167.288,E2 -1167.288} C_VEL
LIN {X 0,Y 594.24,Z 557.201,A -85,B 0,C 180,E1 -1167.966,E2 -1167.966} C_VEL
LIN {X 0,Y 594.239,Z 558.784,A -85,B 0,C 180,E1 -1169.322,E2 -1169.322} C_VEL
LIN {X 0,Y 594.236,Z 559,A -85,B 0,C 180,E1 -1170,E2 -1170} C_VEL
LIN {X 0,Y 594.247,Z 558.185,A -85,B 0,C 180,E1 -1171.355,E2 -1171.355} C_VEL
LIN {X 0,Y 594.24,Z 557.202,A -85,B 0,C 180,E1 -1172.033,E2 -1172.033} C_VEL
LIN {X 0,Y 594.226,Z 555.81,A -85,B 0,C 180,E1 -1172.711,E2 -1172.711} C_VEL
LIN {X 0,Y 594.288,Z 552.897,A -85,B 0,C 180,E1 -1173.729,E2 -1173.729} C_VEL
LIN {X 0,Y 594.241,Z 548.951,A -85,B 0,C 180,E1 -1174.749,E2 -1174.749} C_VEL
LIN {X 0,Y 594.304,Z 542.879,A -85,B 0,C 180,E1 -1175.939,E2 -1175.939} C_VEL
LIN {X 0,Y 594.307,Z 536.238,A -85,B 0,C 180,E1 -1176.962,E2 -1176.962} C_VEL
LIN {X 0,Y 594.359,Z 527.992,A -85,B 0,C 180,E1 -1177.986,E2 -1177.986} C_VEL
LIN {X 0,Y 594.404,Z 517.604,A -85,B 0,C 180,E1 -1179.013,E2 -1179.013} C_VEL
LIN {X 0,Y 594.448,Z 506.752,A -85,B 0,C 180,E1 -1179.871,E2 -1179.871} C_VEL
LIN {X 0,Y 594.505,Z 495.784,A -85,B 0,C 180,E1 -1180.558,E2 -1180.558} C_VEL
LIN {X 0,Y 594.566,Z 483.561,A -85,B 0,C 180,E1 -1181.158,E2 -1181.158} C_VEL
LIN {X 0,Y 594.564,Z 471.886,A -85,B 0,C 180,E1 -1181.592,E2 -1181.592} C_VEL
LIN {X 0,Y 594.633,Z 459.527,A -85,B 0,C 180,E1 -1181.915,E2 -1181.915} C_VEL
LIN {X 0,Y 594.689,Z 443.761,A -85,B 0,C 180,E1 -1182.152,E2 -1182.152} C_VEL
LIN {X 0,Y 594.622,Z 348.29,A -85,B 0,C 180,E1 -1183.311,E2 -1183.311} C_VEL
LIN {X 0,Y 594.442,Z 346.616,A -85,B 0,C 180,E1 -1183.351,E2 -1183.351} C_VEL
LIN {X 0,Y 594.498,Z 326.066,A -85,B 0,C 180,E1 -1186.129,E2 -1186.129} C_VEL
LIN {X 0,Y 594.606,Z 306.009,A -85,B 0,C 180,E1 -1188.877,E2 -1188.877} C_VEL
LIN {X 0,Y 594.73,Z 284.643,A -85,B 0,C 180,E1 -1191.853,E2 -1191.853} C_VEL
LIN {X 0,Y 594.673,Z 277.926,A -85,B 0,C 180,E1 -1192.805,E2 -1192.805} C_VEL
LIN {X 0,Y 594.391,Z 276.445,A -85,B 0,C 180,E1 -1193.058,E2 -1193.058} C_VEL
LIN {X 0,Y 594.371,Z 276.442,A -85,B 0,C 180,E1 -1195.193,E2 -1195.193} C_VEL
LIN {X 0,Y 594.387,Z 276.442,A -85,B 0,C 180,E1 -1197.526,E2 -1197.526} C_VEL
LIN {X 0,Y 594.386,Z 276.446,A -85,B 0,C 180,E1 -1200.328,E2 -1200.328} C_VEL
LIN {X 0,Y 594.376,Z 276.44,A -85,B 0,C 180,E1 -1202.95,E2 -1202.95} C_VEL
LIN {X 0,Y 594.347,Z 276.444,A -85,B 0,C 180,E1 -1205.409,E2 -1205.409} C_VEL
LIN {X 0,Y 594.384,Z 276.444,A -85,B 0,C 180,E1 -1207.94,E2 -1207.94} C_VEL
LIN {X 0,Y 594.376,Z 276.444,A -85,B 0,C 180,E1 -1210.821,E2 -1210.821} C_VEL
LIN {X 0,Y 594.365,Z 276.442,A -85,B 0,C 180,E1 -1213.299,E2 -1213.299} C_VEL
LIN {X 0,Y 594.357,Z 276.447,A -85,B 0,C 180,E1 -1216.161,E2 -1216.161} C_VEL
LIN {X 0,Y 594.38,Z 276.45,A -85,B 0,C 180,E1 -1218.536,E2 -1218.536} C_VEL
LIN {X 0,Y 594.379,Z 276.441,A -85,B 0,C 180,E1 -1221.295,E2 -1221.295} C_VEL
LIN {X 0,Y 594.358,Z 276.442,A -85,B 0,C 180,E1 -1223.756,E2 -1223.756} C_VEL
LIN {X 0,Y 594.375,Z 276.442,A -85,B 0,C 180,E1 -1226.238,E2 -1226.238} C_VEL
LIN {X 0,Y 594.387,Z 276.446,A -85,B 0,C 180,E1 -1228.651,E2 -1228.651} C_VEL
LIN {X 0,Y 594.378,Z 276.449,A -85,B 0,C 180,E1 -1231.042,E2 -1231.042} C_VEL
LIN {X 0,Y 594.384,Z 276.439,A -85,B 0,C 180,E1 -1233.976,E2 -1233.976} C_VEL
LIN {X 0,Y 594.385,Z 276.439,A -85,B 0,C 180,E1 -1236.296,E2 -1236.296} C_VEL
LIN {X 0,Y 594.399,Z 276.447,A -85,B 0,C 180,E1 -1239.224,E2 -1239.224} C_VEL
LIN {X 0,Y 594.347,Z 276.444,A -85,B 0,C 180,E1 -1242.095,E2 -1242.095} C_VEL
LIN {X 0,Y 594.36,Z 276.442,A -85,B 0,C 180,E1 -1244.219,E2 -1244.219} C_VEL
LIN {X 0,Y 594.365,Z 276.446,A -85,B 0,C 180,E1 -1247.017,E2 -1247.017} C_VEL
LIN {X 0,Y 594.383,Z 276.444,A -85,B 0,C 180,E1 -1249.784,E2 -1249.784} C_VEL
LIN {X 0,Y 594.388,Z 276.438,A -85,B 0,C 180,E1 -1252.527,E2 -1252.527} C_VEL
LIN {X 0,Y 594.392,Z 276.443,A -85,B 0,C 180,E1 -1255.252,E2 -1255.252} C_VEL
LIN {X 0,Y 594.382,Z 276.445,A -85,B 0,C 180,E1 -1257.967,E2 -1257.967} C_VEL
LIN {X 0,Y 594.406,Z 276.436,A -85,B 0,C 180,E1 -1260.677,E2 -1260.677} C_VEL
LIN {X 0,Y 594.385,Z 276.443,A -85,B 0,C 180,E1 -1263.389,E2 -1263.389} C_VEL
LIN {X 0,Y 594.363,Z 276.449,A -85,B 0,C 180,E1 -1266.109,E2 -1266.109} C_VEL
LIN {X 0,Y 594.407,Z 276.444,A -85,B 0,C 180,E1 -1268.157,E2 -1268.157} C_VEL
LIN {X 0,Y 594.374,Z 276.44,A -85,B 0,C 180,E1 -1271.069,E2 -1271.069} C_VEL
LIN {X 0,Y 594.375,Z 276.444,A -85,B 0,C 180,E1 -1273.679,E2 -1273.679} C_VEL
LIN {X 0,Y 594.343,Z 276.444,A -85,B 0,C 180,E1 -1275.308,E2 -1275.308} C_VEL
LIN {X 0,Y 593.678,Z 276.534,A -85,B 0,C 180,E1 -1275.874,E2 -1275.874} C_VEL
LIN {X 0,Y 590.818,Z 276.895,A -85,B 0,C 180,E1 -1276.792,E2 -1276.792} C_VEL
LIN {X 0,Y 588.405,Z 277.197,A -85,B 0,C 180,E1 -1277.531,E2 -1277.531} C_VEL
LIN {X 0,Y 587.378,Z 277.321,A -85,B 0,C 180,E1 -1278.101,E2 -1278.101} C_VEL
LIN {X 0,Y 587.3,Z 277.328,A -85,B 0,C 180,E1 -1278.294,E2 -1278.294} C_VEL
LIN {X 0,Y 587.325,Z 277.319,A -85,B 0,C 180,E1 -1281.038,E2 -1281.038} C_VEL
LIN {X 0,Y 587.309,Z 277.32,A -85,B 0,C 180,E1 -1283.259,E2 -1283.259} C_VEL
LIN {X 0,Y 587.322,Z 277.319,A -85,B 0,C 180,E1 -1285.517,E2 -1285.517} C_VEL
LIN {X 0,Y 587.3,Z 277.323,A -85,B 0,C 180,E1 -1287.82,E2 -1287.82} C_VEL
LIN {X 0,Y 587.329,Z 277.329,A -85,B 0,C 180,E1 -1290.51,E2 -1290.51} C_VEL
LIN {X 0,Y 587.322,Z 277.319,A -85,B 0,C 180,E1 -1293.397,E2 -1293.397} C_VEL
LIN {X 0,Y 587.284,Z 277.324,A -85,B 0,C 180,E1 -1295.9,E2 -1295.9} C_VEL
LIN {X 0,Y 587.321,Z 277.325,A -85,B 0,C 180,E1 -1298.48,E2 -1298.48} C_VEL
LIN {X 0,Y 587.325,Z 277.324,A -85,B 0,C 180,E1 -1301.158,E2 -1301.158} C_VEL
LIN {X 0,Y 587.312,Z 277.32,A -85,B 0,C 180,E1 -1304.113,E2 -1304.113} C_VEL
LIN {X 0,Y 587.295,Z 277.333,A -85,B 0,C 180,E1 -1306.993,E2 -1306.993} C_VEL
LIN {X 0,Y 587.3,Z 277.323,A -85,B 0,C 180,E1 -1309.745,E2 -1309.745} C_VEL
LIN {X 0,Y 587.335,Z 277.318,A -85,B 0,C 180,E1 -1312.392,E2 -1312.392} C_VEL
LIN {X 0,Y 587.333,Z 277.321,A -85,B 0,C 180,E1 -1315.654,E2 -1315.654} C_VEL
LIN {X 0,Y 587.328,Z 277.318,A -85,B 0,C 180,E1 -1318.231,E2 -1318.231} C_VEL
LIN {X 0,Y 587.31,Z 277.332,A -85,B 0,C 180,E1 -1321.403,E2 -1321.403} C_VEL
LIN {X 0,Y 587.292,Z 277.327,A -85,B 0,C 180,E1 -1323.832,E2 -1323.832} C_VEL
LIN {X 0,Y 587.304,Z 277.324,A -85,B 0,C 180,E1 -1325.993,E2 -1325.993} C_VEL
LIN {X 0,Y 587.307,Z 277.322,A -85,B 0,C 180,E1 -1328.226,E2 -1328.226} C_VEL
LIN {X 0,Y 587.343,Z 277.319,A -85,B 0,C 180,E1 -1331.151,E2 -1331.151} C_VEL
LIN {X 0,Y 587.299,Z 277.328,A -85,B 0,C 180,E1 -1334.025,E2 -1334.025} C_VEL
LIN {X 0,Y 587.333,Z 277.323,A -85,B 0,C 180,E1 -1336.154,E2 -1336.154} C_VEL
LIN {X 0,Y 587.289,Z 277.324,A -85,B 0,C 180,E1 -1338.962,E2 -1338.962} C_VEL
LIN {X 0,Y 587.318,Z 277.37,A -85,B 0,C 180,E1 -1341.094,E2 -1341.094} C_VEL
LIN {X 0,Y 587.432,Z 284.893,A -85,B 0,C 180,E1 -1342.438,E2 -1342.438} C_VEL
LIN {X 0,Y 587.347,Z 298.596,A -85,B 0,C 180,E1 -1344.851,E2 -1344.851} C_VEL
LIN {X 0,Y 587.259,Z 308.327,A -85,B 0,C 180,E1 -1346.548,E2 -1346.548} C_VEL
LIN {X 0,Y 587.859,Z 313.147,A -85,B 0,C 180,E1 -1346.638,E2 -1346.638} C_VEL
LIN {X 0,Y 587.694,Z 415.051,A -85,B 0,C 180,E1 -1347.901,E2 -1347.901} C_VEL
LIN {X 0,Y 587.675,Z 428.07,A -85,B 0,C 180,E1 -1348.201,E2 -1348.201} C_VEL
LIN {X 0,Y 587.626,Z 440.611,A -85,B 0,C 180,E1 -1348.63,E2 -1348.63} C_VEL
LIN {X 0,Y 587.515,Z 451.84,A -85,B 0,C 180,E1 -1349.143,E2 -1349.143} C_VEL
LIN {X 0,Y 587.441,Z 463.431,A -85,B 0,C 180,E1 -1349.829,E2 -1349.829} C_VEL
LIN {X 0,Y 587.391,Z 473.833,A -85,B 0,C 180,E1 -1350.6,E2 -1350.6} C_VEL
LIN {X 0,Y 587.338,Z 482.346,A -85,B 0,C 180,E1 -1351.372,E2 -1351.372} C_VEL
LIN {X 0,Y 587.266,Z 490.291,A -85,B 0,C 180,E1 -1352.229,E2 -1352.229} C_VEL
LIN {X 0,Y 587.217,Z 498.071,A -85,B 0,C 180,E1 -1353.259,E2 -1353.259} C_VEL
LIN {X 0,Y 587.186,Z 503.373,A -85,B 0,C 180,E1 -1354.118,E2 -1354.118} C_VEL
LIN {X 0,Y 587.158,Z 508.564,A -85,B 0,C 180,E1 -1355.151,E2 -1355.151} C_VEL
LIN {X 0,Y 587.166,Z 512.603,A -85,B 0,C 180,E1 -1356.184,E2 -1356.184} C_VEL
LIN {X 0,Y 587.164,Z 514.712,A -85,B 0,C 180,E1 -1356.875,E2 -1356.875} C_VEL
LIN {X 0,Y 587.145,Z 516.379,A -85,B 0,C 180,E1 -1357.566,E2 -1357.566} C_VEL
LIN {X 0,Y 587.138,Z 517.638,A -85,B 0,C 180,E1 -1358.259,E2 -1358.259} C_VEL
LIN {X 0,Y 587.127,Z 518.498,A -85,B 0,C 180,E1 -1358.952,E2 -1358.952} C_VEL
LIN {X 0,Y 587.15,Z 518.916,A -85,B 0,C 180,E1 -1359.647,E2 -1359.647} C_VEL
LIN {X 0,Y 587.163,Z 518.572,A -85,B 0,C 180,E1 -1361.041,E2 -1361.041} C_VEL
LIN {X 0,Y 587.153,Z 517.782,A -85,B 0,C 180,E1 -1361.741,E2 -1361.741} C_VEL
LIN {X 0,Y 587.161,Z 516.549,A -85,B 0,C 180,E1 -1362.442,E2 -1362.442} C_VEL
LIN {X 0,Y 587.156,Z 513.89,A -85,B 0,C 180,E1 -1363.498,E2 -1363.498} C_VEL
LIN {X 0,Y 587.189,Z 510.164,A -85,B 0,C 180,E1 -1364.557,E2 -1364.557} C_VEL
LIN {X 0,Y 587.192,Z 505.243,A -85,B 0,C 180,E1 -1365.623,E2 -1365.623} C_VEL
LIN {X 0,Y 587.236,Z 498.415,A -85,B 0,C 180,E1 -1366.777,E2 -1366.777} C_VEL
LIN {X 0,Y 587.305,Z 491.083,A -85,B 0,C 180,E1 -1367.767,E2 -1367.767} C_VEL
LIN {X 0,Y 587.335,Z 482.838,A -85,B 0,C 180,E1 -1368.668,E2 -1368.668} C_VEL
LIN {X 0,Y 587.353,Z 474.7,A -85,B 0,C 180,E1 -1369.419,E2 -1369.419} C_VEL
LIN {X 0,Y 587.42,Z 464.188,A -85,B 0,C 180,E1 -1370.21,E2 -1370.21} C_VEL
LIN {X 0,Y 587.52,Z 453.674,A -85,B 0,C 180,E1 -1370.847,E2 -1370.847} C_VEL
LIN {X 0,Y 587.602,Z 441.928,A -85,B 0,C 180,E1 -1371.409,E2 -1371.409} C_VEL
LIN {X 0,Y 587.623,Z 429.285,A -85,B 0,C 180,E1 -1371.855,E2 -1371.855} C_VEL
LIN {X 0,Y 587.631,Z 416.877,A -85,B 0,C 180,E1 -1372.155,E2 -1372.155} C_VEL
LIN {X 0,Y 587.707,Z 392.947,A -85,B 0,C 180,E1 -1372.476,E2 -1372.476} C_VEL
LIN {X 0,Y 587.806,Z 311.429,A -85,B 0,C 180,E1 -1373.475,E2 -1373.475} C_VEL
LIN {X 0,Y 587.299,Z 308.331,A -85,B 0,C 180,E1 -1373.54,E2 -1373.54} C_VEL
LIN {X 0,Y 587.362,Z 295.108,A -85,B 0,C 180,E1 -1375.85,E2 -1375.85} C_VEL
LIN {X 0,Y 587.495,Z 279.621,A -85,B 0,C 180,E1 -1378.588,E2 -1378.588} C_VEL
LIN {X 0,Y 587.387,Z 277.315,A -85,B 0,C 180,E1 -1379.035,E2 -1379.035} C_VEL
LIN {X 0,Y 587.344,Z 277.321,A -85,B 0,C 180,E1 -1381.836,E2 -1381.836} C_VEL
LIN {X 0,Y 587.341,Z 277.328,A -85,B 0,C 180,E1 -1384.347,E2 -1384.347} C_VEL
LIN {X 0,Y 587.343,Z 277.316,A -85,B 0,C 180,E1 -1387.608,E2 -1387.608} C_VEL
LIN {X 0,Y 587.311,Z 277.327,A -85,B 0,C 180,E1 -1390.255,E2 -1390.255} C_VEL
LIN {X 0,Y 587.314,Z 277.323,A -85,B 0,C 180,E1 -1393.118,E2 -1393.118} C_VEL
LIN {X 0,Y 587.311,Z 277.322,A -85,B 0,C 180,E1 -1396.048,E2 -1396.048} C_VEL
LIN {X 0,Y 587.335,Z 277.326,A -85,B 0,C 180,E1 -1398.925,E2 -1398.925} C_VEL
LIN {X 0,Y 587.328,Z 277.319,A -85,B 0,C 180,E1 -1401.521,E2 -1401.521} C_VEL
LIN {X 0,Y 587.29,Z 277.323,A -85,B 0,C 180,E1 -1404.1,E2 -1404.1} C_VEL
LIN {X 0,Y 587.331,Z 277.321,A -85,B 0,C 180,E1 -1406.603,E2 -1406.603} C_VEL
LIN {X 0,Y 587.336,Z 277.321,A -85,B 0,C 180,E1 -1409.49,E2 -1409.49} C_VEL
LIN {X 0,Y 587.35,Z 277.315,A -85,B 0,C 180,E1 -1412.307,E2 -1412.307} C_VEL
LIN {X 0,Y 587.331,Z 277.318,A -85,B 0,C 180,E1 -1414.483,E2 -1414.483} C_VEL
LIN {X 0,Y 587.317,Z 277.326,A -85,B 0,C 180,E1 -1417.131,E2 -1417.131} C_VEL
LIN {X 0,Y 587.328,Z 277.323,A -85,B 0,C 180,E1 -1419.695,E2 -1419.695} C_VEL
LIN {X 0,Y 587.307,Z 277.325,A -85,B 0,C 180,E1 -1421.873,E2 -1421.873} C_VEL
LIN {X 0,Y 587.322,Z 277.321,A -85,B 0,C 180,E1 -1424.025,E2 -1424.025} C_VEL
LIN {X 0,Y 587.357,Z 277.317,A -85,B 0,C 180,E1 -1426.154,E2 -1426.154} C_VEL
LIN {X 0,Y 587.337,Z 277.317,A -85,B 0,C 180,E1 -1428.962,E2 -1428.962} C_VEL
LIN {X 0,Y 587.362,Z 277.325,A -85,B 0,C 180,E1 -1431.745,E2 -1431.745} C_VEL
LIN {X 0,Y 587.357,Z 277.316,A -85,B 0,C 180,E1 -1434.507,E2 -1434.507} C_VEL
LIN {X 0,Y 587.367,Z 277.314,A -85,B 0,C 180,E1 -1437.257,E2 -1437.257} C_VEL
LIN {X 0,Y 587.382,Z 277.322,A -85,B 0,C 180,E1 -1440,E2 -1440} C_VEL
LIN {X 0,Y 587.369,Z 277.314,A -85,B 0,C 180,E1 -1442.743,E2 -1442.743} C_VEL
LIN {X 0,Y 587.356,Z 277.315,A -85,B 0,C 180,E1 -1445.493,E2 -1445.493} C_VEL
LIN {X 0,Y 587.362,Z 277.324,A -85,B 0,C 180,E1 -1448.255,E2 -1448.255} C_VEL
LIN {X 0,Y 587.348,Z 277.315,A -85,B 0,C 180,E1 -1451.134,E2 -1451.134} C_VEL
LIN {X 0,Y 587.364,Z 277.321,A -85,B 0,C 180,E1 -1454.261,E2 -1454.261} C_VEL
LIN {X 0,Y 587.347,Z 277.316,A -85,B 0,C 180,E1 -1457.406,E2 -1457.406} C_VEL
LIN {X 0,Y 587.313,Z 277.32,A -85,B 0,C 180,E1 -1459.576,E2 -1459.576} C_VEL
LIN {X 0,Y 587.338,Z 277.324,A -85,B 0,C 180,E1 -1462.514,E2 -1462.514} C_VEL
LIN {X 0,Y 587.351,Z 277.326,A -85,B 0,C 180,E1 -1464.759,E2 -1464.759} C_VEL
LIN {X 0,Y 587.329,Z 277.326,A -85,B 0,C 180,E1 -1467.046,E2 -1467.046} C_VEL
LIN {X 0,Y 587.346,Z 277.319,A -85,B 0,C 180,E1 -1469.38,E2 -1469.38} C_VEL
LIN {X 0,Y 587.342,Z 277.316,A -85,B 0,C 180,E1 -1471.836,E2 -1471.836} C_VEL
LIN {X 0,Y 587.347,Z 277.316,A -85,B 0,C 180,E1 -1474.348,E2 -1474.348} C_VEL
LIN {X 0,Y 587.346,Z 277.32,A -85,B 0,C 180,E1 -1477.608,E2 -1477.608} C_VEL
LIN {X 0,Y 587.312,Z 277.318,A -85,B 0,C 180,E1 -1480.255,E2 -1480.255} C_VEL
LIN {X 0,Y 587.317,Z 277.326,A -85,B 0,C 180,E1 -1483.119,E2 -1483.119} C_VEL
LIN {X 0,Y 587.313,Z 277.322,A -85,B 0,C 180,E1 -1486.049,E2 -1486.049} C_VEL
LIN {X 0,Y 587.337,Z 277.319,A -85,B 0,C 180,E1 -1488.925,E2 -1488.925} C_VEL
LIN {X 0,Y 587.327,Z 277.328,A -85,B 0,C 180,E1 -1491.521,E2 -1491.521} C_VEL
LIN {X 0,Y 587.291,Z 277.327,A -85,B 0,C 180,E1 -1494.1,E2 -1494.1} C_VEL
LIN {X 0,Y 587.329,Z 277.319,A -85,B 0,C 180,E1 -1496.603,E2 -1496.603} C_VEL
LIN {X 0,Y 587.339,Z 277.322,A -85,B 0,C 180,E1 -1499.49,E2 -1499.49} C_VEL
LIN {X 0,Y 587.344,Z 277.321,A -85,B 0,C 180,E1 -1502.309,E2 -1502.309} C_VEL
LIN {X 0,Y 587.35,Z 277.317,A -85,B 0,C 180,E1 -1505.241,E2 -1505.241} C_VEL
LIN {X 0,Y 587.356,Z 277.418,A -85,B 0,C 180,E1 -1506.821,E2 -1506.821} C_VEL
LIN {X 0,Y 587.859,Z 280.915,A -85,B 0,C 180,E1 -1507.344,E2 -1507.344} C_VEL
LIN {X 0,Y 587.698,Z 300.173,A -85,B 0,C 180,E1 -1510.073,E2 -1510.073} C_VEL
LIN {X 0,Y 587.568,Z 319.453,A -85,B 0,C 180,E1 -1512.761,E2 -1512.761} C_VEL
LIN {X 0,Y 587.451,Z 341.887,A -85,B 0,C 180,E1 -1515.843,E2 -1515.843} C_VEL
LIN {X 0,Y 587.392,Z 346.612,A -85,B 0,C 180,E1 -1516.486,E2 -1516.486} C_VEL
LIN {X 0,Y 587.87,Z 350.709,A -85,B 0,C 180,E1 -1516.563,E2 -1516.563} C_VEL
LIN {X 0,Y 587.725,Z 454.939,A -85,B 0,C 180,E1 -1517.855,E2 -1517.855} C_VEL
LIN {X 0,Y 587.672,Z 468.214,A -85,B 0,C 180,E1 -1518.16,E2 -1518.16} C_VEL
LIN {X 0,Y 587.603,Z 480.619,A -85,B 0,C 180,E1 -1518.584,E2 -1518.584} C_VEL
LIN {X 0,Y 587.549,Z 492.628,A -85,B 0,C 180,E1 -1519.141,E2 -1519.141} C_VEL
LIN {X 0,Y 587.443,Z 504.2,A -85,B 0,C 180,E1 -1519.836,E2 -1519.836} C_VEL
LIN {X 0,Y 587.392,Z 514.596,A -85,B 0,C 180,E1 -1520.618,E2 -1520.618} C_VEL
LIN {X 0,Y 587.299,Z 523.041,A -85,B 0,C 180,E1 -1521.397,E2 -1521.397} C_VEL
LIN {X 0,Y 587.274,Z 530.959,A -85,B 0,C 180,E1 -1522.263,E2 -1522.263} C_VEL
LIN {X 0,Y 587.23,Z 537.468,A -85,B 0,C 180,E1 -1523.126,E2 -1523.126} C_VEL
LIN {X 0,Y 587.236,Z 543.865,A -85,B 0,C 180,E1 -1524.161,E2 -1524.161} C_VEL
LIN {X 0,Y 587.147,Z 548.949,A -85,B 0,C 180,E1 -1525.193,E2 -1525.193} C_VEL
LIN {X 0,Y 587.212,Z 552.895,A -85,B 0,C 180,E1 -1526.225,E2 -1526.225} C_VEL
LIN {X 0,Y 587.132,Z 555.808,A -85,B 0,C 180,E1 -1527.255,E2 -1527.255} C_VEL
LIN {X 0,Y 587.139,Z 557.2,A -85,B 0,C 180,E1 -1527.942,E2 -1527.942} C_VEL
LIN {X 0,Y 587.14,Z 558.784,A -85,B 0,C 180,E1 -1529.314,E2 -1529.314} C_VEL
LIN {X 0,Y 587.137,Z 559,A -85,B 0,C 180,E1 -1530,E2 -1530} C_VEL
LIN {X 0,Y 587.147,Z 558.186,A -85,B 0,C 180,E1 -1531.372,E2 -1531.372} C_VEL
LIN {X 0,Y 587.139,Z 557.201,A -85,B 0,C 180,E1 -1532.058,E2 -1532.058} C_VEL
LIN {X 0,Y 587.132,Z 555.81,A -85,B 0,C 180,E1 -1532.744,E2 -1532.744} C_VEL
LIN {X 0,Y 587.212,Z 552.897,A -85,B 0,C 180,E1 -1533.774,E2 -1533.774} C_VEL
LIN {X 0,Y 587.147,Z 548.951,A -85,B 0,C 180,E1 -1534.806,E2 -1534.806} C_VEL
LIN {X 0,Y 587.217,Z 542.879,A -85,B 0,C 180,E1 -1536.011,E2 -1536.011} C_VEL
LIN {X 0,Y 587.244,Z 536.239,A -85,B 0,C 180,E1 -1537.046,E2 -1537.046} C_VEL
LIN {X 0,Y 587.297,Z 527.993,A -85,B 0,C 180,E1 -1538.083,E2 -1538.083} C_VEL
LIN {X 0,Y 587.357,Z 517.605,A -85,B 0,C 180,E1 -1539.122,E2 -1539.122} C_VEL
LIN {X 0,Y 587.444,Z 506.752,A -85,B 0,C 180,E1 -1539.989,E2 -1539.989} C_VEL
LIN {X 0,Y 587.521,Z 495.786,A -85,B 0,C 180,E1 -1540.685,E2 -1540.685} C_VEL
LIN {X 0,Y 587.602,Z 483.797,A -85,B 0,C 180,E1 -1541.282,E2 -1541.282} C_VEL
LIN {X 0,Y 587.617,Z 471.884,A -85,B 0,C 180,E1 -1541.731,E2 -1541.731} C_VEL
LIN {X 0,Y 587.688,Z 459.526,A -85,B 0,C 180,E1 -1542.058,E2 -1542.058} C_VEL
LIN {X 0,Y 587.744,Z 443.761,A -85,B 0,C 180,E1 -1542.298,E2 -1542.298} C_VEL
LIN {X 0,Y 587.719,Z 348.736,A -85,B 0,C 180,E1 -1543.465,E2 -1543.465} C_VEL
LIN {X 0,Y 587.392,Z 346.616,A -85,B 0,C 180,E1 -1543.514,E2 -1543.514} C_VEL
LIN {X 0,Y 587.47,Z 328.655,A -85,B 0,C 180,E1 -1545.971,E2 -1545.971} C_VEL
LIN {X 0,Y 587.632,Z 309.238,A -85,B 0,C 180,E1 -1548.658,E2 -1548.658} C_VEL
LIN {X 0,Y 587.802,Z 288.501,A -85,B 0,C 180,E1 -1551.575,E2 -1551.575} C_VEL
LIN {X 0,Y 587.806,Z 279.777,A -85,B 0,C 180,E1 -1552.821,E2 -1552.821} C_VEL
LIN {X 0,Y 587.335,Z 277.325,A -85,B 0,C 180,E1 -1553.205,E2 -1553.205} C_VEL
LIN {X 0,Y 587.33,Z 277.323,A -85,B 0,C 180,E1 -1555.516,E2 -1555.516} C_VEL
LIN {X 0,Y 587.347,Z 277.323,A -85,B 0,C 180,E1 -1557.817,E2 -1557.817} C_VEL
LIN {X 0,Y 587.337,Z 277.321,A -85,B 0,C 180,E1 -1560.509,E2 -1560.509} C_VEL
LIN {X 0,Y 587.332,Z 277.318,A -85,B 0,C 180,E1 -1563.396,E2 -1563.396} C_VEL
LIN {X 0,Y 587.29,Z 277.328,A -85,B 0,C 180,E1 -1565.9,E2 -1565.9} C_VEL
LIN {X 0,Y 587.327,Z 277.326,A -85,B 0,C 180,E1 -1568.479,E2 -1568.479} C_VEL
LIN {X 0,Y 587.335,Z 277.318,A -85,B 0,C 180,E1 -1571.156,E2 -1571.156} C_VEL
LIN {X 0,Y 587.31,Z 277.325,A -85,B 0,C 180,E1 -1574.111,E2 -1574.111} C_VEL
LIN {X 0,Y 587.313,Z 277.323,A -85,B 0,C 180,E1 -1576.993,E2 -1576.993} C_VEL
LIN {X 0,Y 587.31,Z 277.32,A -85,B 0,C 180,E1 -1579.745,E2 -1579.745} C_VEL
LIN {X 0,Y 587.343,Z 277.322,A -85,B 0,C 180,E1 -1582.392,E2 -1582.392} C_VEL
LIN {X 0,Y 587.344,Z 277.316,A -85,B 0,C 180,E1 -1585.652,E2 -1585.652} C_VEL
LIN {X 0,Y 587.348,Z 277.317,A -85,B 0,C 180,E1 -1588.231,E2 -1588.231} C_VEL
LIN {X 0,Y 587.345,Z 277.326,A -85,B 0,C 180,E1 -1590.866,E2 -1590.866} C_VEL
LIN {X 0,Y 587.356,Z 277.315,A -85,B 0,C 180,E1 -1593.818,E2 -1593.818} C_VEL
LIN {X 0,Y 587.332,Z 277.318,A -85,B 0,C 180,E1 -1595.993,E2 -1595.993} C_VEL
LIN {X 0,Y 587.315,Z 277.32,A -85,B 0,C 180,E1 -1598.225,E2 -1598.225} C_VEL
LIN {X 0,Y 587.345,Z 277.326,A -85,B 0,C 180,E1 -1601.151,E2 -1601.151} C_VEL
LIN {X 0,Y 587.317,Z 277.32,A -85,B 0,C 180,E1 -1604.024,E2 -1604.024} C_VEL
LIN {X 0,Y 587.353,Z 277.315,A -85,B 0,C 180,E1 -1606.154,E2 -1606.154} C_VEL
LIN {X 0,Y 587.34,Z 277.32,A -85,B 0,C 180,E1 -1608.962,E2 -1608.962} C_VEL
LIN {X 0,Y 587.362,Z 277.32,A -85,B 0,C 180,E1 -1611.745,E2 -1611.745} C_VEL
LIN {X 0,Y 587.352,Z 277.315,A -85,B 0,C 180,E1 -1614.507,E2 -1614.507} C_VEL
LIN {X 0,Y 587.373,Z 277.317,A -85,B 0,C 180,E1 -1617.257,E2 -1617.257} C_VEL
LIN {X 0,Y 587.372,Z 277.319,A -85,B 0,C 180,E1 -1620,E2 -1620} C_VEL
LIN {X 0,Y 587.36,Z 277.314,A -85,B 0,C 180,E1 -1622.743,E2 -1622.743} C_VEL
LIN {X 0,Y 587.36,Z 277.318,A -85,B 0,C 180,E1 -1625.493,E2 -1625.493} C_VEL
LIN {X 0,Y 587.358,Z 277.32,A -85,B 0,C 180,E1 -1628.255,E2 -1628.255} C_VEL
LIN {X 0,Y 587.342,Z 277.316,A -85,B 0,C 180,E1 -1631.134,E2 -1631.134} C_VEL
LIN {X 0,Y 587.352,Z 277.321,A -85,B 0,C 180,E1 -1633.846,E2 -1633.846} C_VEL
LIN {X 0,Y 587.334,Z 277.319,A -85,B 0,C 180,E1 -1636.811,E2 -1636.811} C_VEL
LIN {X 0,Y 587.3,Z 277.328,A -85,B 0,C 180,E1 -1638.294,E2 -1638.294} C_VEL
LIN {X 0,Y 586.654,Z 277.404,A -85,B 0,C 180,E1 -1638.866,E2 -1638.866} C_VEL
LIN {X 0,Y 583.833,Z 277.757,A -85,B 0,C 180,E1 -1639.794,E2 -1639.794} C_VEL
LIN {X 0,Y 581.426,Z 278.06,A -85,B 0,C 180,E1 -1640.541,E2 -1640.541} C_VEL
LIN {X 0,Y 580.373,Z 278.185,A -85,B 0,C 180,E1 -1641.118,E2 -1641.118} C_VEL
LIN {X 0,Y 580.278,Z 278.196,A -85,B 0,C 180,E1 -1641.313,E2 -1641.313} C_VEL
LIN {X 0,Y 580.292,Z 278.204,A -85,B 0,C 180,E1 -1644.316,E2 -1644.316} C_VEL
LIN {X 0,Y 580.263,Z 278.206,A -85,B 0,C 180,E1 -1646.624,E2 -1646.624} C_VEL
LIN {X 0,Y 580.291,Z 278.195,A -85,B 0,C 180,E1 -1649.309,E2 -1649.309} C_VEL
LIN {X 0,Y 580.293,Z 278.199,A -85,B 0,C 180,E1 -1652.201,E2 -1652.201} C_VEL
LIN {X 0,Y 580.282,Z 278.207,A -85,B 0,C 180,E1 -1654.697,E2 -1654.697} C_VEL
LIN {X 0,Y 580.291,Z 278.197,A -85,B 0,C 180,E1 -1657.269,E2 -1657.269} C_VEL
LIN {X 0,Y 580.282,Z 278.198,A -85,B 0,C 180,E1 -1660.27,E2 -1660.27} C_VEL
LIN {X 0,Y 580.269,Z 278.205,A -85,B 0,C 180,E1 -1662.707,E2 -1662.707} C_VEL
LIN {X 0,Y 580.253,Z 278.201,A -85,B 0,C 180,E1 -1665.611,E2 -1665.611} C_VEL
LIN {X 0,Y 580.269,Z 278.202,A -85,B 0,C 180,E1 -1668.67,E2 -1668.67} C_VEL
LIN {X 0,Y 580.265,Z 278.206,A -85,B 0,C 180,E1 -1670.965,E2 -1670.965} C_VEL
LIN {X 0,Y 580.262,Z 278.202,A -85,B 0,C 180,E1 -1673.597,E2 -1673.597} C_VEL
LIN {X 0,Y 580.273,Z 278.197,A -85,B 0,C 180,E1 -1676.143,E2 -1676.143} C_VEL
LIN {X 0,Y 580.261,Z 278.199,A -85,B 0,C 180,E1 -1678.614,E2 -1678.614} C_VEL
LIN {X 0,Y 580.281,Z 278.2,A -85,B 0,C 180,E1 -1681.024,E2 -1681.024} C_VEL
LIN {X 0,Y 580.243,Z 278.202,A -85,B 0,C 180,E1 -1684.149,E2 -1684.149} C_VEL
LIN {X 0,Y 580.257,Z 278.201,A -85,B 0,C 180,E1 -1686.999,E2 -1686.999} C_VEL
LIN {X 0,Y 580.268,Z 278.205,A -85,B 0,C 180,E1 -1689.437,E2 -1689.437} C_VEL
LIN {X 0,Y 580.253,Z 278.21,A -85,B 0,C 180,E1 -1691.645,E2 -1691.645} C_VEL
LIN {X 0,Y 580.275,Z 278.197,A -85,B 0,C 180,E1 -1694.547,E2 -1694.547} C_VEL
LIN {X 0,Y 580.245,Z 278.201,A -85,B 0,C 180,E1 -1696.696,E2 -1696.696} C_VEL
LIN {X 0,Y 580.266,Z 278.199,A -85,B 0,C 180,E1 -1698.826,E2 -1698.826} C_VEL
LIN {X 0,Y 580.272,Z 278.33,A -85,B 0,C 180,E1 -1701.029,E2 -1701.029} C_VEL
LIN {X 0,Y 580.483,Z 283.652,A -85,B 0,C 180,E1 -1701.997,E2 -1701.997} C_VEL
LIN {X 0,Y 580.327,Z 299.305,A -85,B 0,C 180,E1 -1704.789,E2 -1704.789} C_VEL
LIN {X 0,Y 580.24,Z 308.417,A -85,B 0,C 180,E1 -1706.398,E2 -1706.398} C_VEL
LIN {X 0,Y 580.962,Z 314.25,A -85,B 0,C 180,E1 -1706.489,E2 -1706.489} C_VEL
LIN {X 0,Y 580.773,Z 414.618,A -85,B 0,C 180,E1 -1707.746,E2 -1707.746} C_VEL
LIN {X 0,Y 580.72,Z 427.804,A -85,B 0,C 180,E1 -1708.05,E2 -1708.05} C_VEL
LIN {X 0,Y 580.677,Z 440.409,A -85,B 0,C 180,E1 -1708.483,E2 -1708.483} C_VEL
LIN {X 0,Y 580.518,Z 452.516,A -85,B 0,C 180,E1 -1709.046,E2 -1709.046} C_VEL
LIN {X 0,Y 580.42,Z 463.958,A -85,B 0,C 180,E1 -1709.74,E2 -1709.74} C_VEL
LIN {X 0,Y 580.36,Z 474.269,A -85,B 0,C 180,E1 -1710.521,E2 -1710.521} C_VEL
LIN {X 0,Y 580.291,Z 483.549,A -85,B 0,C 180,E1 -1711.388,E2 -1711.388} C_VEL
LIN {X 0,Y 580.205,Z 491.311,A -85,B 0,C 180,E1 -1712.256,E2 -1712.256} C_VEL
LIN {X 0,Y 580.127,Z 498.861,A -85,B 0,C 180,E1 -1713.299,E2 -1713.299} C_VEL
LIN {X 0,Y 580.118,Z 505.853,A -85,B 0,C 180,E1 -1714.517,E2 -1714.517} C_VEL
LIN {X 0,Y 580.117,Z 510.508,A -85,B 0,C 180,E1 -1715.562,E2 -1715.562} C_VEL
LIN {X 0,Y 580.107,Z 513.958,A -85,B 0,C 180,E1 -1716.572,E2 -1716.572} C_VEL
LIN {X 0,Y 580.065,Z 516.633,A -85,B 0,C 180,E1 -1717.659,E2 -1717.659} C_VEL
LIN {X 0,Y 580.059,Z 517.833,A -85,B 0,C 180,E1 -1718.36,E2 -1718.36} C_VEL
LIN {X 0,Y 580.026,Z 518.59,A -85,B 0,C 180,E1 -1719.063,E2 -1719.063} C_VEL
LIN {X 0,Y 580.056,Z 518.944,A -85,B 0,C 180,E1 -1719.766,E2 -1719.766} C_VEL
LIN {X 0,Y 580.07,Z 518.556,A -85,B 0,C 180,E1 -1721.075,E2 -1721.075} C_VEL
LIN {X 0,Y 580.053,Z 517.585,A -85,B 0,C 180,E1 -1721.887,E2 -1721.887} C_VEL
LIN {X 0,Y 580.054,Z 516.289,A -85,B 0,C 180,E1 -1722.597,E2 -1722.597} C_VEL
LIN {X 0,Y 580.072,Z 513.508,A -85,B 0,C 180,E1 -1723.666,E2 -1723.666} C_VEL
LIN {X 0,Y 580.125,Z 509.649,A -85,B 0,C 180,E1 -1724.739,E2 -1724.739} C_VEL
LIN {X 0,Y 580.135,Z 504.584,A -85,B 0,C 180,E1 -1725.818,E2 -1725.818} C_VEL
LIN {X 0,Y 580.179,Z 498.149,A -85,B 0,C 180,E1 -1726.901,E2 -1726.901} C_VEL
LIN {X 0,Y 580.212,Z 489.992,A -85,B 0,C 180,E1 -1727.992,E2 -1727.992} C_VEL
LIN {X 0,Y 580.27,Z 481.581,A -85,B 0,C 180,E1 -1728.904,E2 -1728.904} C_VEL
LIN {X 0,Y 580.397,Z 471.228,A -85,B 0,C 180,E1 -1729.819,E2 -1729.819} C_VEL
LIN {X 0,Y 580.439,Z 460.824,A -85,B 0,C 180,E1 -1730.557,E2 -1730.557} C_VEL
LIN {X 0,Y 580.593,Z 448.633,A -85,B 0,C 180,E1 -1731.24,E2 -1731.24} C_VEL
LIN {X 0,Y 580.613,Z 436.568,A -85,B 0,C 180,E1 -1731.759,E2 -1731.759} C_VEL
LIN {X 0,Y 580.674,Z 423.147,A -85,B 0,C 180,E1 -1732.165,E2 -1732.165} C_VEL
LIN {X 0,Y 580.71,Z 410.313,A -85,B 0,C 180,E1 -1732.41,E2 -1732.41} C_VEL
LIN {X 0,Y 580.83,Z 311.779,A -85,B 0,C 180,E1 -1733.635,E2 -1733.635} C_VEL
LIN {X 0,Y 580.267,Z 308.366,A -85,B 0,C 180,E1 -1733.7,E2 -1733.7} C_VEL
LIN {X 0,Y 580.374,Z 293.398,A -85,B 0,C 180,E1 -1736.35,E2 -1736.35} C_VEL
LIN {X 0,Y 580.483,Z 279.911,A -85,B 0,C 180,E1 -1738.768,E2 -1738.768} C_VEL
LIN {X 0,Y 580.352,Z 278.192,A -85,B 0,C 180,E1 -1739.093,E2 -1739.093} C_VEL
LIN {X 0,Y 580.298,Z 278.205,A -85,B 0,C 180,E1 -1742.201,E2 -1742.201} C_VEL
LIN {X 0,Y 580.286,Z 278.201,A -85,B 0,C 180,E1 -1744.696,E2 -1744.696} C_VEL
LIN {X 0,Y 580.297,Z 278.193,A -85,B 0,C 180,E1 -1747.268,E2 -1747.268} C_VEL
LIN {X 0,Y 580.29,Z 278.202,A -85,B 0,C 180,E1 -1750.27,E2 -1750.27} C_VEL
LIN {X 0,Y 580.276,Z 278.206,A -85,B 0,C 180,E1 -1752.706,E2 -1752.706} C_VEL
LIN {X 0,Y 580.254,Z 278.2,A -85,B 0,C 180,E1 -1755.611,E2 -1755.611} C_VEL
LIN {X 0,Y 580.28,Z 278.199,A -85,B 0,C 180,E1 -1758.231,E2 -1758.231} C_VEL
LIN {X 0,Y 580.278,Z 278.205,A -85,B 0,C 180,E1 -1760.965,E2 -1760.965} C_VEL
LIN {X 0,Y 580.267,Z 278.198,A -85,B 0,C 180,E1 -1763.596,E2 -1763.596} C_VEL
LIN {X 0,Y 580.314,Z 278.191,A -85,B 0,C 180,E1 -1766.145,E2 -1766.145} C_VEL
LIN {X 0,Y 580.274,Z 278.2,A -85,B 0,C 180,E1 -1768.615,E2 -1768.615} C_VEL
LIN {X 0,Y 580.291,Z 278.203,A -85,B 0,C 180,E1 -1771.024,E2 -1771.024} C_VEL
LIN {X 0,Y 580.29,Z 278.198,A -85,B 0,C 180,E1 -1773.666,E2 -1773.666} C_VEL
LIN {X 0,Y 580.299,Z 278.197,A -85,B 0,C 180,E1 -1775.684,E2 -1775.684} C_VEL
LIN {X 0,Y 580.27,Z 278.199,A -85,B 0,C 180,E1 -1777.947,E2 -1777.947} C_VEL
LIN {X 0,Y 580.299,Z 278.195,A -85,B 0,C 180,E1 -1780.914,E2 -1780.914} C_VEL
LIN {X 0,Y 580.277,Z 278.202,A -85,B 0,C 180,E1 -1783.826,E2 -1783.826} C_VEL
LIN {X 0,Y 580.324,Z 278.195,A -85,B 0,C 180,E1 -1785.983,E2 -1785.983} C_VEL
LIN {X 0,Y 580.304,Z 278.193,A -85,B 0,C 180,E1 -1788.827,E2 -1788.827} C_VEL
LIN {X 0,Y 580.326,Z 278.199,A -85,B 0,C 180,E1 -1791.644,E2 -1791.644} C_VEL
LIN {X 0,Y 580.322,Z 278.193,A -85,B 0,C 180,E1 -1794.44,E2 -1794.44} C_VEL
LIN {X 0,Y 580.334,Z 278.19,A -85,B 0,C 180,E1 -1797.224,E2 -1797.224} C_VEL
LIN {X 0,Y 580.352,Z 278.197,A -85,B 0,C 180,E1 -1800,E2 -1800} C_VEL
LIN {X 0,Y 580.336,Z 278.19,A -85,B 0,C 180,E1 -1802.777,E2 -1802.777} C_VEL
LIN {X 0,Y 580.322,Z 278.192,A -85,B 0,C 180,E1 -1805.56,E2 -1805.56} C_VEL
LIN {X 0,Y 580.326,Z 278.2,A -85,B 0,C 180,E1 -1808.356,E2 -1808.356} C_VEL
LIN {X 0,Y 580.3,Z 278.193,A -85,B 0,C 180,E1 -1811.191,E2 -1811.191} C_VEL
LIN {X 0,Y 580.325,Z 278.194,A -85,B 0,C 180,E1 -1814.017,E2 -1814.017} C_VEL
LIN {X 0,Y 580.312,Z 278.197,A -85,B 0,C 180,E1 -1816.914,E2 -1816.914} C_VEL
LIN {X 0,Y 580.287,Z 278.195,A -85,B 0,C 180,E1 -1819.823,E2 -1819.823} C_VEL
LIN {X 0,Y 580.268,Z 278.199,A -85,B 0,C 180,E1 -1822.053,E2 -1822.053} C_VEL
LIN {X 0,Y 580.306,Z 278.199,A -85,B 0,C 180,E1 -1825.08,E2 -1825.08} C_VEL
LIN {X 0,Y 580.298,Z 278.194,A -85,B 0,C 180,E1 -1828.186,E2 -1828.186} C_VEL
LIN {X 0,Y 580.284,Z 278.201,A -85,B 0,C 180,E1 -1830.695,E2 -1830.695} C_VEL
LIN {X 0,Y 580.302,Z 278.2,A -85,B 0,C 180,E1 -1833.316,E2 -1833.316} C_VEL
LIN {X 0,Y 580.245,Z 278.201,A -85,B 0,C 180,E1 -1835.756,E2 -1835.756} C_VEL
LIN {X 0,Y 580.288,Z 278.195,A -85,B 0,C 180,E1 -1838.147,E2 -1838.147} C_VEL
LIN {X 0,Y 580.298,Z 278.195,A -85,B 0,C 180,E1 -1840.844,E2 -1840.844} C_VEL
LIN {X 0,Y 580.274,Z 278.203,A -85,B 0,C 180,E1 -1843.659,E2 -1843.659} C_VEL
LIN {X 0,Y 580.275,Z 278.197,A -85,B 0,C 180,E1 -1846.61,E2 -1846.61} C_VEL
LIN {X 0,Y 580.299,Z 278.198,A -85,B 0,C 180,E1 -1849.157,E2 -1849.157} C_VEL
LIN {X 0,Y 580.29,Z 278.2,A -85,B 0,C 180,E1 -1851.927,E2 -1851.927} C_VEL
LIN {X 0,Y 580.251,Z 278.201,A -85,B 0,C 180,E1 -1854.453,E2 -1854.453} C_VEL
LIN {X 0,Y 580.29,Z 278.196,A -85,B 0,C 180,E1 -1856.975,E2 -1856.975} C_VEL
LIN {X 0,Y 580.298,Z 278.198,A -85,B 0,C 180,E1 -1859.425,E2 -1859.425} C_VEL
LIN {X 0,Y 580.294,Z 278.203,A -85,B 0,C 180,E1 -1862.143,E2 -1862.143} C_VEL
LIN {X 0,Y 580.323,Z 278.193,A -85,B 0,C 180,E1 -1865.27,E2 -1865.27} C_VEL
LIN {X 0,Y 580.31,Z 278.259,A -85,B 0,C 180,E1 -1866.659,E2 -1866.659} C_VEL
LIN {X 0,Y 580.935,Z 283.345,A -85,B 0,C 180,E1 -1867.412,E2 -1867.412} C_VEL
LIN {X 0,Y 580.752,Z 302.762,A -85,B 0,C 180,E1 -1870.194,E2 -1870.194} C_VEL
LIN {X 0,Y 580.57,Z 322.716,A -85,B 0,C 180,E1 -1873.004,E2 -1873.004} C_VEL
LIN {X 0,Y 580.423,Z 345.479,A -85,B 0,C 180,E1 -1876.164,E2 -1876.164} C_VEL
LIN {X 0,Y 580.398,Z 346.612,A -85,B 0,C 180,E1 -1876.32,E2 -1876.32} C_VEL
LIN {X 0,Y 580.987,Z 352.498,A -85,B 0,C 180,E1 -1876.423,E2 -1876.423} C_VEL
LIN {X 0,Y 580.787,Z 454.939,A -85,B 0,C 180,E1 -1877.708,E2 -1877.708} C_VEL
LIN {X 0,Y 580.73,Z 468.214,A -85,B 0,C 180,E1 -1878.017,E2 -1878.017} C_VEL
LIN {X 0,Y 580.628,Z 480.37,A -85,B 0,C 180,E1 -1878.435,E2 -1878.435} C_VEL
LIN {X 0,Y 580.556,Z 492.626,A -85,B 0,C 180,E1 -1879.008,E2 -1879.008} C_VEL
LIN {X 0,Y 580.421,Z 504.2,A -85,B 0,C 180,E1 -1879.712,E2 -1879.712} C_VEL
LIN {X 0,Y 580.343,Z 514.598,A -85,B 0,C 180,E1 -1880.503,E2 -1880.503} C_VEL
LIN {X 0,Y 580.263,Z 523.054,A -85,B 0,C 180,E1 -1881.292,E2 -1881.292} C_VEL
LIN {X 0,Y 580.222,Z 530.959,A -85,B 0,C 180,E1 -1882.168,E2 -1882.168} C_VEL
LIN {X 0,Y 580.156,Z 538.635,A -85,B 0,C 180,E1 -1883.219,E2 -1883.219} C_VEL
LIN {X 0,Y 580.139,Z 545.679,A -85,B 0,C 180,E1 -1884.438,E2 -1884.438} C_VEL
LIN {X 0,Y 580.108,Z 550.371,A -85,B 0,C 180,E1 -1885.483,E2 -1885.483} C_VEL
LIN {X 0,Y 580.123,Z 553.956,A -85,B 0,C 180,E1 -1886.527,E2 -1886.527} C_VEL
LIN {X 0,Y 580.043,Z 555.808,A -85,B 0,C 180,E1 -1887.222,E2 -1887.222} C_VEL
LIN {X 0,Y 580.038,Z 557.198,A -85,B 0,C 180,E1 -1887.917,E2 -1887.917} C_VEL
LIN {X 0,Y 580.04,Z 558.785,A -85,B 0,C 180,E1 -1889.306,E2 -1889.306} C_VEL
LIN {X 0,Y 580.037,Z 559,A -85,B 0,C 180,E1 -1890,E2 -1890} C_VEL
LIN {X 0,Y 580.046,Z 558.186,A -85,B 0,C 180,E1 -1891.388,E2 -1891.388} C_VEL
LIN {X 0,Y 580.038,Z 557.2,A -85,B 0,C 180,E1 -1892.083,E2 -1892.083} C_VEL
LIN {X 0,Y 580.043,Z 555.81,A -85,B 0,C 180,E1 -1892.778,E2 -1892.778} C_VEL
LIN {X 0,Y 580.109,Z 552.897,A -85,B 0,C 180,E1 -1893.82,E2 -1893.82} C_VEL
LIN {X 0,Y 580.053,Z 548.95,A -85,B 0,C 180,E1 -1894.865,E2 -1894.865} C_VEL
LIN {X 0,Y 580.14,Z 542.879,A -85,B 0,C 180,E1 -1896.084,E2 -1896.084} C_VEL
LIN {X 0,Y 580.184,Z 536.24,A -85,B 0,C 180,E1 -1897.132,E2 -1897.132} C_VEL
LIN {X 0,Y 580.246,Z 527.993,A -85,B 0,C 180,E1 -1898.182,E2 -1898.182} C_VEL
LIN {X 0,Y 580.332,Z 517.605,A -85,B 0,C 180,E1 -1899.233,E2 -1899.233} C_VEL
LIN {X 0,Y 580.43,Z 507.931,A -85,B 0,C 180,E1 -1900.023,E2 -1900.023} C_VEL
LIN {X 0,Y 580.531,Z 497.333,A -85,B 0,C 180,E1 -1900.727,E2 -1900.727} C_VEL
LIN {X 0,Y 580.613,Z 485.487,A -85,B 0,C 180,E1 -1901.344,E2 -1901.344} C_VEL
LIN {X 0,Y 580.652,Z 473.183,A -85,B 0,C 180,E1 -1901.829,E2 -1901.829} C_VEL
LIN {X 0,Y 580.755,Z 460.534,A -85,B 0,C 180,E1 -1902.182,E2 -1902.182} C_VEL
LIN {X 0,Y 580.834,Z 447.339,A -85,B 0,C 180,E1 -1902.402,E2 -1902.402} C_VEL
LIN {X 0,Y 580.805,Z 349.409,A -85,B 0,C 180,E1 -1903.62,E2 -1903.62} C_VEL
LIN {X 0,Y 580.398,Z 346.616,A -85,B 0,C 180,E1 -1903.68,E2 -1903.68} C_VEL
LIN {X 0,Y 580.544,Z 326.066,A -85,B 0,C 180,E1 -1906.528,E2 -1906.528} C_VEL
LIN {X 0,Y 580.753,Z 305.067,A -85,B 0,C 180,E1 -1909.479,E2 -1909.479} C_VEL
LIN {X 0,Y 580.966,Z 284.643,A -85,B 0,C 180,E1 -1912.399,E2 -1912.399} C_VEL
LIN {X 0,Y 580.635,Z 279.959,A -85,B 0,C 180,E1 -1913.088,E2 -1913.088} C_VEL
LIN {X 0,Y 580.312,Z 278.201,A -85,B 0,C 180,E1 -1913.377,E2 -1913.377} C_VEL
LIN {X 0,Y 580.281,Z 278.206,A -85,B 0,C 180,E1 -1915.849,E2 -1915.849} C_VEL
LIN {X 0,Y 580.299,Z 278.203,A -85,B 0,C 180,E1 -1918.185,E2 -1918.185} C_VEL
LIN {X 0,Y 580.284,Z 278.197,A -85,B 0,C 180,E1 -1920.694,E2 -1920.694} C_VEL
LIN {X 0,Y 580.302,Z 278.193,A -85,B 0,C 180,E1 -1923.316,E2 -1923.316} C_VEL
LIN {X 0,Y 580.244,Z 278.203,A -85,B 0,C 180,E1 -1925.756,E2 -1925.756} C_VEL
LIN {X 0,Y 580.286,Z 278.203,A -85,B 0,C 180,E1 -1928.146,E2 -1928.146} C_VEL
LIN {X 0,Y 580.297,Z 278.197,A -85,B 0,C 180,E1 -1930.843,E2 -1930.843} C_VEL
LIN {X 0,Y 580.271,Z 278.198,A -85,B 0,C 180,E1 -1933.658,E2 -1933.658} C_VEL
LIN {X 0,Y 580.272,Z 278.207,A -85,B 0,C 180,E1 -1936.609,E2 -1936.609} C_VEL
LIN {X 0,Y 580.296,Z 278.196,A -85,B 0,C 180,E1 -1939.156,E2 -1939.156} C_VEL
LIN {X 0,Y 580.287,Z 278.196,A -85,B 0,C 180,E1 -1941.926,E2 -1941.926} C_VEL
LIN {X 0,Y 580.251,Z 278.205,A -85,B 0,C 180,E1 -1944.452,E2 -1944.452} C_VEL
LIN {X 0,Y 580.287,Z 278.203,A -85,B 0,C 180,E1 -1946.975,E2 -1946.975} C_VEL
LIN {X 0,Y 580.299,Z 278.196,A -85,B 0,C 180,E1 -1949.425,E2 -1949.425} C_VEL
LIN {X 0,Y 580.294,Z 278.194,A -85,B 0,C 180,E1 -1952.141,E2 -1952.141} C_VEL
LIN {X 0,Y 580.317,Z 278.198,A -85,B 0,C 180,E1 -1955.269,E2 -1955.269} C_VEL
LIN {X 0,Y 580.266,Z 278.198,A -85,B 0,C 180,E1 -1957.947,E2 -1957.947} C_VEL
LIN {X 0,Y 580.314,Z 278.198,A -85,B 0,C 180,E1 -1960.914,E2 -1960.914} C_VEL
LIN {X 0,Y 580.272,Z 278.199,A -85,B 0,C 180,E1 -1963.825,E2 -1963.825} C_VEL
LIN {X 0,Y 580.32,Z 278.193,A -85,B 0,C 180,E1 -1965.983,E2 -1965.983} C_VEL
LIN {X 0,Y 580.299,Z 278.195,A -85,B 0,C 180,E1 -1968.827,E2 -1968.827} C_VEL
LIN {X 0,Y 580.327,Z 278.199,A -85,B 0,C 180,E1 -1971.644,E2 -1971.644} C_VEL
LIN {X 0,Y 580.317,Z 278.192,A -85,B 0,C 180,E1 -1974.44,E2 -1974.44} C_VEL
LIN {X 0,Y 580.339,Z 278.192,A -85,B 0,C 180,E1 -1977.223,E2 -1977.223} C_VEL
LIN {X 0,Y 580.342,Z 278.194,A -85,B 0,C 180,E1 -1980,E2 -1980} C_VEL
LIN {X 0,Y 580.328,Z 278.19,A -85,B 0,C 180,E1 -1982.776,E2 -1982.776} C_VEL
LIN {X 0,Y 580.324,Z 278.196,A -85,B 0,C 180,E1 -1985.56,E2 -1985.56} C_VEL
LIN {X 0,Y 580.321,Z 278.195,A -85,B 0,C 180,E1 -1988.356,E2 -1988.356} C_VEL
LIN {X 0,Y 580.294,Z 278.194,A -85,B 0,C 180,E1 -1991.191,E2 -1991.191} C_VEL
LIN {X 0,Y 580.309,Z 278.202,A -85,B 0,C 180,E1 -1994.017,E2 -1994.017} C_VEL
LIN {X 0,Y 580.306,Z 278.194,A -85,B 0,C 180,E1 -1996.914,E2 -1996.914} C_VEL
LIN {X 0,Y 580.281,Z 278.199,A -85,B 0,C 180,E1 -1999.823,E2 -1999.823} C_VEL
LIN {X 0,Y 580.278,Z 278.196,A -85,B 0,C 180,E1 -2001.313,E2 -2001.313} C_VEL
LIN {X 0,Y 579.579,Z 278.289,A -85,B 0,C 180,E1 -2001.892,E2 -2001.892} C_VEL
LIN {X 0,Y 576.7,Z 278.645,A -85,B 0,C 180,E1 -2002.832,E2 -2002.832} C_VEL
LIN {X 0,Y 574.306,Z 278.942,A -85,B 0,C 180,E1 -2003.588,E2 -2003.588} C_VEL
LIN {X 0,Y 573.307,Z 279.072,A -85,B 0,C 180,E1 -2004.172,E2 -2004.172} C_VEL
LIN {X 0,Y 573.24,Z 279.077,A -85,B 0,C 180,E1 -2004.37,E2 -2004.37} C_VEL
LIN {X 0,Y 573.199,Z 279.081,A -85,B 0,C 180,E1 -2006.978,E2 -2006.978} C_VEL
LIN {X 0,Y 573.237,Z 279.073,A -85,B 0,C 180,E1 -2009.488,E2 -2009.488} C_VEL
LIN {X 0,Y 573.247,Z 279.083,A -85,B 0,C 180,E1 -2012.645,E2 -2012.645} C_VEL
LIN {X 0,Y 573.2,Z 279.081,A -85,B 0,C 180,E1 -2015.188,E2 -2015.188} C_VEL
LIN {X 0,Y 573.228,Z 279.074,A -85,B 0,C 180,E1 -2017.808,E2 -2017.808} C_VEL
LIN {X 0,Y 573.24,Z 279.079,A -85,B 0,C 180,E1 -2020.525,E2 -2020.525} C_VEL
LIN {X 0,Y 573.226,Z 279.078,A -85,B 0,C 180,E1 -2023.36,E2 -2023.36} C_VEL
LIN {X 0,Y 573.231,Z 279.075,A -85,B 0,C 180,E1 -2026.332,E2 -2026.332} C_VEL
LIN {X 0,Y 573.241,Z 279.077,A -85,B 0,C 180,E1 -2029.475,E2 -2029.475} C_VEL
LIN {X 0,Y 573.226,Z 279.075,A -85,B 0,C 180,E1 -2032.192,E2 -2032.192} C_VEL
LIN {X 0,Y 573.229,Z 279.086,A -85,B 0,C 180,E1 -2035.229,E2 -2035.229} C_VEL
LIN {X 0,Y 573.231,Z 279.074,A -85,B 0,C 180,E1 -2038.185,E2 -2038.185} C_VEL
LIN {X 0,Y 573.23,Z 279.075,A -85,B 0,C 180,E1 -2040.633,E2 -2040.633} C_VEL
LIN {X 0,Y 573.197,Z 279.089,A -85,B 0,C 180,E1 -2043.516,E2 -2043.516} C_VEL
LIN {X 0,Y 573.206,Z 279.079,A -85,B 0,C 180,E1 -2046.134,E2 -2046.134} C_VEL
LIN {X 0,Y 573.249,Z 279.072,A -85,B 0,C 180,E1 -2048.71,E2 -2048.71} C_VEL
LIN {X 0,Y 573.211,Z 279.083,A -85,B 0,C 180,E1 -2051.411,E2 -2051.411} C_VEL
LIN {X 0,Y 573.216,Z 279.078,A -85,B 0,C 180,E1 -2054.352,E2 -2054.352} C_VEL
LIN {X 0,Y 573.206,Z 279.079,A -85,B 0,C 180,E1 -2056.529,E2 -2056.529} C_VEL
LIN {X 0,Y 573.237,Z 279.078,A -85,B 0,C 180,E1 -2059.403,E2 -2059.403} C_VEL
LIN {X 0,Y 573.234,Z 279.168,A -85,B 0,C 180,E1 -2060.94,E2 -2060.94} C_VEL
LIN {X 0,Y 573.476,Z 284.363,A -85,B 0,C 180,E1 -2061.898,E2 -2061.898} C_VEL
LIN {X 0,Y 573.307,Z 300.014,A -85,B 0,C 180,E1 -2064.725,E2 -2064.725} C_VEL
LIN {X 0,Y 573.225,Z 308.385,A -85,B 0,C 180,E1 -2066.222,E2 -2066.222} C_VEL
LIN {X 0,Y 574.062,Z 313.621,A -85,B 0,C 180,E1 -2066.315,E2 -2066.315} C_VEL
LIN {X 0,Y 573.833,Z 415.348,A -85,B 0,C 180,E1 -2067.609,E2 -2067.609} C_VEL
LIN {X 0,Y 573.764,Z 429.031,A -85,B 0,C 180,E1 -2067.938,E2 -2067.938} C_VEL
LIN {X 0,Y 573.699,Z 441.321,A -85,B 0,C 180,E1 -2068.377,E2 -2068.377} C_VEL
LIN {X 0,Y 573.529,Z 453.158,A -85,B 0,C 180,E1 -2068.947,E2 -2068.947} C_VEL
LIN {X 0,Y 573.399,Z 464.485,A -85,B 0,C 180,E1 -2069.649,E2 -2069.649} C_VEL
LIN {X 0,Y 573.329,Z 474.705,A -85,B 0,C 180,E1 -2070.439,E2 -2070.439} C_VEL
LIN {X 0,Y 573.24,Z 483.073,A -85,B 0,C 180,E1 -2071.23,E2 -2071.23} C_VEL
LIN {X 0,Y 573.132,Z 490.902,A -85,B 0,C 180,E1 -2072.108,E2 -2072.108} C_VEL
LIN {X 0,Y 573.077,Z 498.533,A -85,B 0,C 180,E1 -2073.164,E2 -2073.164} C_VEL
LIN {X 0,Y 573.035,Z 504.685,A -85,B 0,C 180,E1 -2074.22,E2 -2074.22} C_VEL
LIN {X 0,Y 572.997,Z 509.589,A -85,B 0,C 180,E1 -2075.278,E2 -2075.278} C_VEL
LIN {X 0,Y 573.027,Z 514.074,A -85,B 0,C 180,E1 -2076.568,E2 -2076.568} C_VEL
LIN {X 0,Y 572.975,Z 516.888,A -85,B 0,C 180,E1 -2077.754,E2 -2077.754} C_VEL
LIN {X 0,Y 572.949,Z 517.988,A -85,B 0,C 180,E1 -2078.465,E2 -2078.465} C_VEL
LIN {X 0,Y 572.972,Z 518.971,A -85,B 0,C 180,E1 -2079.888,E2 -2079.888} C_VEL
LIN {X 0,Y 572.982,Z 518.538,A -85,B 0,C 180,E1 -2081.113,E2 -2081.113} C_VEL
LIN {X 0,Y 572.947,Z 517.386,A -85,B 0,C 180,E1 -2082.036,E2 -2082.036} C_VEL
LIN {X 0,Y 572.951,Z 516.026,A -85,B 0,C 180,E1 -2082.756,E2 -2082.756} C_VEL
LIN {X 0,Y 572.992,Z 513.122,A -85,B 0,C 180,E1 -2083.838,E2 -2083.838} C_VEL
LIN {X 0,Y 573.029,Z 509.13,A -85,B 0,C 180,E1 -2084.925,E2 -2084.925} C_VEL
LIN {X 0,Y 573.089,Z 502.904,A -85,B 0,C 180,E1 -2086.2,E2 -2086.2} C_VEL
LIN {X 0,Y 573.123,Z 496.001,A -85,B 0,C 180,E1 -2087.3,E2 -2087.3} C_VEL
LIN {X 0,Y 573.198,Z 487.337,A -85,B 0,C 180,E1 -2088.404,E2 -2088.404} C_VEL
LIN {X 0,Y 573.277,Z 477.278,A -85,B 0,C 180,E1 -2089.423,E2 -2089.423} C_VEL
LIN {X 0,Y 573.388,Z 467.061,A -85,B 0,C 180,E1 -2090.259,E2 -2090.259} C_VEL
LIN {X 0,Y 573.51,Z 456.289,A -85,B 0,C 180,E1 -2090.966,E2 -2090.966} C_VEL
LIN {X 0,Y 573.648,Z 443.655,A -85,B 0,C 180,E1 -2091.611,E2 -2091.611} C_VEL
LIN {X 0,Y 573.718,Z 431.397,A -85,B 0,C 180,E1 -2092.081,E2 -2092.081} C_VEL
LIN {X 0,Y 573.736,Z 418.935,A -85,B 0,C 180,E1 -2092.412,E2 -2092.412} C_VEL
LIN {X 0,Y 573.839,Z 401.868,A -85,B 0,C 180,E1 -2092.669,E2 -2092.669} C_VEL
LIN {X 0,Y 573.967,Z 312.846,A -85,B 0,C 180,E1 -2093.787,E2 -2093.787} C_VEL
LIN {X 0,Y 573.231,Z 308.399,A -85,B 0,C 180,E1 -2093.866,E2 -2093.866} C_VEL
LIN {X 0,Y 573.376,Z 293.59,A -85,B 0,C 180,E1 -2096.52,E2 -2096.52} C_VEL
LIN {X 0,Y 573.445,Z 280.198,A -85,B 0,C 180,E1 -2098.954,E2 -2098.954} C_VEL
LIN {X 0,Y 573.3,Z 279.071,A -85,B 0,C 180,E1 -2099.213,E2 -2099.213} C_VEL
LIN {X 0,Y 573.251,Z 279.083,A -85,B 0,C 180,E1 -2102.228,E2 -2102.228} C_VEL
LIN {X 0,Y 573.233,Z 279.078,A -85,B 0,C 180,E1 -2104.771,E2 -2104.771} C_VEL
LIN {X 0,Y 573.233,Z 279.075,A -85,B 0,C 180,E1 -2107.808,E2 -2107.808} C_VEL
LIN {X 0,Y 573.244,Z 279.084,A -85,B 0,C 180,E1 -2110.525,E2 -2110.525} C_VEL
LIN {X 0,Y 573.236,Z 279.075,A -85,B 0,C 180,E1 -2113.359,E2 -2113.359} C_VEL
LIN {X 0,Y 573.237,Z 279.084,A -85,B 0,C 180,E1 -2116.641,E2 -2116.641} C_VEL
LIN {X 0,Y 573.243,Z 279.074,A -85,B 0,C 180,E1 -2119.475,E2 -2119.475} C_VEL
LIN {X 0,Y 573.235,Z 279.074,A -85,B 0,C 180,E1 -2122.192,E2 -2122.192} C_VEL
LIN {X 0,Y 573.235,Z 279.079,A -85,B 0,C 180,E1 -2125.228,E2 -2125.228} C_VEL
LIN {X 0,Y 573.249,Z 279.072,A -85,B 0,C 180,E1 -2127.772,E2 -2127.772} C_VEL
LIN {X 0,Y 573.263,Z 279.072,A -85,B 0,C 180,E1 -2130.634,E2 -2130.634} C_VEL
LIN {X 0,Y 573.249,Z 279.078,A -85,B 0,C 180,E1 -2133.024,E2 -2133.024} C_VEL
LIN {X 0,Y 573.273,Z 279.077,A -85,B 0,C 180,E1 -2135.366,E2 -2135.366} C_VEL
LIN {X 0,Y 573.227,Z 279.074,A -85,B 0,C 180,E1 -2138.419,E2 -2138.419} C_VEL
LIN {X 0,Y 573.267,Z 279.069,A -85,B 0,C 180,E1 -2140.731,E2 -2140.731} C_VEL
LIN {X 0,Y 573.249,Z 279.081,A -85,B 0,C 180,E1 -2143.622,E2 -2143.622} C_VEL
LIN {X 0,Y 573.272,Z 279.076,A -85,B 0,C 180,E1 -2145.807,E2 -2145.807} C_VEL
LIN {X 0,Y 573.262,Z 279.07,A -85,B 0,C 180,E1 -2148.745,E2 -2148.745} C_VEL
LIN {X 0,Y 573.282,Z 279.075,A -85,B 0,C 180,E1 -2151.541,E2 -2151.541} C_VEL
LIN {X 0,Y 573.288,Z 279.07,A -85,B 0,C 180,E1 -2154.372,E2 -2154.372} C_VEL
LIN {X 0,Y 573.311,Z 279.074,A -85,B 0,C 180,E1 -2157.893,E2 -2157.893} C_VEL
LIN {X 0,Y 573.328,Z 279.063,A -85,B 0,C 180,E1 -2160.703,E2 -2160.703} C_VEL
LIN {X 0,Y 573.235,Z 279.074,A -85,B 0,C 180,E1 -2163.515,E2 -2163.515} C_VEL
LIN {X 0,Y 573.288,Z 279.069,A -85,B 0,C 180,E1 -2165.628,E2 -2165.628} C_VEL
LIN {X 0,Y 573.282,Z 279.076,A -85,B 0,C 180,E1 -2168.46,E2 -2168.46} C_VEL
LIN {X 0,Y 573.271,Z 279.068,A -85,B 0,C 180,E1 -2171.312,E2 -2171.312} C_VEL
LIN {X 0,Y 573.281,Z 279.078,A -85,B 0,C 180,E1 -2174.425,E2 -2174.425} C_VEL
LIN {X 0,Y 573.258,Z 279.073,A -85,B 0,C 180,E1 -2177.112,E2 -2177.112} C_VEL
LIN {X 0,Y 573.242,Z 279.074,A -85,B 0,C 180,E1 -2180.077,E2 -2180.077} C_VEL
LIN {X 0,Y 573.234,Z 279.078,A -85,B 0,C 180,E1 -2182.338,E2 -2182.338} C_VEL
LIN {X 0,Y 573.254,Z 279.073,A -85,B 0,C 180,E1 -2185.41,E2 -2185.41} C_VEL
LIN {X 0,Y 573.251,Z 279.072,A -85,B 0,C 180,E1 -2188.029,E2 -2188.029} C_VEL
LIN {X 0,Y 573.246,Z 279.073,A -85,B 0,C 180,E1 -2190.176,E2 -2190.176} C_VEL
LIN {X 0,Y 573.253,Z 279.075,A -85,B 0,C 180,E1 -2192.645,E2 -2192.645} C_VEL
LIN {X 0,Y 573.207,Z 279.086,A -85,B 0,C 180,E1 -2195.188,E2 -2195.188} C_VEL
LIN {X 0,Y 573.236,Z 279.075,A -85,B 0,C 180,E1 -2197.808,E2 -2197.808} C_VEL
LIN {X 0,Y 573.245,Z 279.07,A -85,B 0,C 180,E1 -2200.525,E2 -2200.525} C_VEL
LIN {X 0,Y 573.238,Z 279.084,A -85,B 0,C 180,E1 -2203.359,E2 -2203.359} C_VEL
LIN {X 0,Y 573.237,Z 279.074,A -85,B 0,C 180,E1 -2206.641,E2 -2206.641} C_VEL
LIN {X 0,Y 573.246,Z 279.082,A -85,B 0,C 180,E1 -2209.475,E2 -2209.475} C_VEL
LIN {X 0,Y 573.236,Z 279.075,A -85,B 0,C 180,E1 -2212.193,E2 -2212.193} C_VEL
LIN {X 0,Y 573.235,Z 279.077,A -85,B 0,C 180,E1 -2215.229,E2 -2215.229} C_VEL
LIN {X 0,Y 573.252,Z 279.082,A -85,B 0,C 180,E1 -2217.772,E2 -2217.772} C_VEL
LIN {X 0,Y 573.265,Z 279.072,A -85,B 0,C 180,E1 -2220.634,E2 -2220.634} C_VEL
LIN {X 0,Y 573.237,Z 279.077,A -85,B 0,C 180,E1 -2223.508,E2 -2223.508} C_VEL
LIN {X 0,Y 573.238,Z 279.084,A -85,B 0,C 180,E1 -2226.135,E2 -2226.135} C_VEL
LIN {X 0,Y 573.258,Z 279.146,A -85,B 0,C 180,E1 -2226.526,E2 -2226.526} C_VEL
LIN {X 0,Y 573.999,Z 284.423,A -85,B 0,C 180,E1 -2227.314,E2 -2227.314} C_VEL
LIN {X 0,Y 573.833,Z 302.762,A -85,B 0,C 180,E1 -2229.945,E2 -2229.945} C_VEL
LIN {X 0,Y 573.587,Z 323.473,A -85,B 0,C 180,E1 -2232.898,E2 -2232.898} C_VEL
LIN {X 0,Y 573.431,Z 344.185,A -85,B 0,C 180,E1 -2235.811,E2 -2235.811} C_VEL
LIN {X 0,Y 573.393,Z 346.612,A -85,B 0,C 180,E1 -2236.149,E2 -2236.149} C_VEL
LIN {X 0,Y 574.111,Z 352.498,A -85,B 0,C 180,E1 -2236.257,E2 -2236.257} C_VEL
LIN {X 0,Y 573.866,Z 454.939,A -85,B 0,C 180,E1 -2237.557,E2 -2237.557} C_VEL
LIN {X 0,Y 573.789,Z 468.214,A -85,B 0,C 180,E1 -2237.869,E2 -2237.869} C_VEL
LIN {X 0,Y 573.675,Z 480.371,A -85,B 0,C 180,E1 -2238.293,E2 -2238.293} C_VEL
LIN {X 0,Y 573.591,Z 492.632,A -85,B 0,C 180,E1 -2238.874,E2 -2238.874} C_VEL
LIN {X 0,Y 573.437,Z 504.198,A -85,B 0,C 180,E1 -2239.585,E2 -2239.585} C_VEL
LIN {X 0,Y 573.329,Z 514.599,A -85,B 0,C 180,E1 -2240.385,E2 -2240.385} C_VEL
LIN {X 0,Y 573.237,Z 523.068,A -85,B 0,C 180,E1 -2241.184,E2 -2241.184} C_VEL
LIN {X 0,Y 573.16,Z 530.959,A -85,B 0,C 180,E1 -2242.071,E2 -2242.071} C_VEL
LIN {X 0,Y 573.075,Z 538.94,A -85,B 0,C 180,E1 -2243.183,E2 -2243.183} C_VEL
LIN {X 0,Y 573.07,Z 545.679,A -85,B 0,C 180,E1 -2244.369,E2 -2244.369} C_VEL
LIN {X 0,Y 573.028,Z 550.371,A -85,B 0,C 180,E1 -2245.427,E2 -2245.427} C_VEL
LIN {X 0,Y 573.022,Z 553.957,A -85,B 0,C 180,E1 -2246.484,E2 -2246.484} C_VEL
LIN {X 0,Y 572.959,Z 555.808,A -85,B 0,C 180,E1 -2247.187,E2 -2247.187} C_VEL
